    CONST robtarget p4016:= [[1554.6419767101188, 10.164661639834293, 993.500033578516], [0, 0, 1, 0], [0, 0, 0, 0], [9E9, 9E9, 9E9, 9E9, 9E9, 9E9]];
    CONST robtarget p4017:= [[1554.7008352009186, 9.837821442717242, 993.500033578516], [0, 0, 1, 0], [0, 0, 0, 0], [9E9, 9E9, 9E9, 9E9, 9E9, 9E9]];
    CONST robtarget p4018:= [[1554.7242404677872, 9.706052723327417, 993.500033578516], [0, 0, 1, 0], [0, 0, 0, 0], [9E9, 9E9, 9E9, 9E9, 9E9, 9E9]];
    CONST robtarget p4019:= [[1554.7649214276712, 9.482909780103284, 993.500033578516], [0, 0, 1, 0], [0, 0, 0, 0], [9E9, 9E9, 9E9, 9E9, 9E9, 9E9]];
    CONST robtarget p4020:= [[1554.8352270948067, 9.068291490106276, 993.500033578516], [0, 0, 1, 0], [0, 0, 0, 0], [9E9, 9E9, 9E9, 9E9, 9E9, 9E9]];
    CONST robtarget p4021:= [[1554.9212712484702, 8.59744226106804, 993.500033578516], [0, 0, 1, 0], [0, 0, 0, 0], [9E9, 9E9, 9E9, 9E9, 9E9, 9E9]];
    CONST robtarget p4022:= [[1555.0185066025715, 8.144599417769001, 993.500033578516], [0, 0, 1, 0], [0, 0, 0, 0], [9E9, 9E9, 9E9, 9E9, 9E9, 9E9]];
    CONST robtarget p4023:= [[1555.0385939462196, 7.9852680304157815, 993.500033578516], [0, 0, 1, 0], [0, 0, 0, 0], [9E9, 9E9, 9E9, 9E9, 9E9, 9E9]];
    CONST robtarget p4024:= [[1555.0668408502406, 7.720577334258238, 993.500033578516], [0, 0, 1, 0], [0, 0, 0, 0], [9E9, 9E9, 9E9, 9E9, 9E9, 9E9]];
    CONST robtarget p4025:= [[1555.1038402589074, 7.394988314848419, 993.500033578516], [0, 0, 1, 0], [0, 0, 0, 0], [9E9, 9E9, 9E9, 9E9, 9E9, 9E9]];
    CONST robtarget p4026:= [[1555.1141702872178, 7.2850707768797065, 993.500033578516], [0, 0, 1, 0], [0, 0, 0, 0], [9E9, 9E9, 9E9, 9E9, 9E9, 9E9]];
    CONST robtarget p4027:= [[1555.160055171739, 6.884447981356743, 993.500033578516], [0, 0, 1, 0], [0, 0, 0, 0], [9E9, 9E9, 9E9, 9E9, 9E9, 9E9]];
    CONST robtarget p4028:= [[1555.1886068304418, 6.5967447173674145, 993.500033578516], [0, 0, 1, 0], [0, 0, 0, 0], [9E9, 9E9, 9E9, 9E9, 9E9, 9E9]];
    CONST robtarget p4029:= [[1555.2302397704561, 6.209649884868298, 993.500033578516], [0, 0, 1, 0], [0, 0, 0, 0], [9E9, 9E9, 9E9, 9E9, 9E9, 9E9]];
    CONST robtarget p4030:= [[1555.3072534316846, 5.36442871184876, 993.500033578516], [0, 0, 1, 0], [0, 0, 0, 0], [9E9, 9E9, 9E9, 9E9, 9E9, 9E9]];
    CONST robtarget p4031:= [[1555.37826504701, 4.761405763737287, 993.500033578516], [0, 0, 1, 0], [0, 0, 0, 0], [9E9, 9E9, 9E9, 9E9, 9E9, 9E9]];
    CONST robtarget p4032:= [[1555.3863462726958, 4.670605801933405, 993.500033578516], [0, 0, 1, 0], [0, 0, 0, 0], [9E9, 9E9, 9E9, 9E9, 9E9, 9E9]];
    CONST robtarget p4033:= [[1555.4282420152724, 4.316200343407104, 993.500033578516], [0, 0, 1, 0], [0, 0, 0, 0], [9E9, 9E9, 9E9, 9E9, 9E9, 9E9]];
    CONST robtarget p4034:= [[1555.474795687078, 3.9231101854634716, 993.500033578516], [0, 0, 1, 0], [0, 0, 0, 0], [9E9, 9E9, 9E9, 9E9, 9E9, 9E9]];
    CONST robtarget p4035:= [[1555.4964332564984, 3.210495643507869, 993.500033578516], [0, 0, 1, 0], [0, 0, 0, 0], [9E9, 9E9, 9E9, 9E9, 9E9, 9E9]];
    CONST robtarget p4036:= [[1555.4992750024937, 3.001332927943622, 993.500033578516], [0, 0, 1, 0], [0, 0, 0, 0], [9E9, 9E9, 9E9, 9E9, 9E9, 9E9]];
    CONST robtarget p4037:= [[1555.5146870542724, 2.606860948282204, 993.500033578516], [0, 0, 1, 0], [0, 0, 0, 0], [9E9, 9E9, 9E9, 9E9, 9E9, 9E9]];
    CONST robtarget p4038:= [[1555.5401059955102, 2.158807079297702, 993.500033578516], [0, 0, 1, 0], [0, 0, 0, 0], [9E9, 9E9, 9E9, 9E9, 9E9, 9E9]];
    CONST robtarget p4039:= [[1555.5457042027897, 1.9240824141459996, 993.500033578516], [0, 0, 1, 0], [0, 0, 0, 0], [9E9, 9E9, 9E9, 9E9, 9E9, 9E9]];
    CONST robtarget p4040:= [[1555.5560129677121, 1.6442269998726573, 993.500033578516], [0, 0, 1, 0], [0, 0, 0, 0], [9E9, 9E9, 9E9, 9E9, 9E9, 9E9]];
    CONST robtarget p4041:= [[1555.5620302267785, 1.4813565941546756, 993.500033578516], [0, 0, 1, 0], [0, 0, 0, 0], [9E9, 9E9, 9E9, 9E9, 9E9, 9E9]];
    CONST robtarget p4042:= [[1555.569137398368, 1.3324889484946993, 993.500033578516], [0, 0, 1, 0], [0, 0, 0, 0], [9E9, 9E9, 9E9, 9E9, 9E9, 9E9]];
    CONST robtarget p4043:= [[1555.5836986010872, 0.9039823076832789, 993.500033578516], [0, 0, 1, 0], [0, 0, 0, 0], [9E9, 9E9, 9E9, 9E9, 9E9, 9E9]];
    CONST robtarget p4044:= [[1555.584302450153, 0.8259278887639994, 993.500033578516], [0, 0, 1, 0], [0, 0, 0, 0], [9E9, 9E9, 9E9, 9E9, 9E9, 9E9]];
    CONST robtarget p4045:= [[1555.5904849739145, 0.5579150837128566, 993.500033578516], [0, 0, 1, 0], [0, 0, 0, 0], [9E9, 9E9, 9E9, 9E9, 9E9, 9E9]];
    CONST robtarget p4046:= [[1555.6069058610203, 0.01192725742885159, 993.500033578516], [0, 0, 1, 0], [0, 0, 0, 0], [9E9, 9E9, 9E9, 9E9, 9E9, 9E9]];
    CONST robtarget p4047:= [[1555.6080018663752, -0.28272944407356704, 993.500033578516], [0, 0, 1, 0], [0, 0, 0, 0], [9E9, 9E9, 9E9, 9E9, 9E9, 9E9]];
    CONST robtarget p4048:= [[1555.5897069092575, -0.568370675110188, 993.500033578516], [0, 0, 1, 0], [0, 0, 0, 0], [9E9, 9E9, 9E9, 9E9, 9E9, 9E9]];
    CONST robtarget p4049:= [[1555.5753783303503, -1.0723405994250186, 993.500033578516], [0, 0, 1, 0], [0, 0, 0, 0], [9E9, 9E9, 9E9, 9E9, 9E9, 9E9]];
    CONST robtarget p4050:= [[1555.5457633836807, -1.5150721807046637, 993.500033578516], [0, 0, 1, 0], [0, 0, 0, 0], [9E9, 9E9, 9E9, 9E9, 9E9, 9E9]];
    CONST robtarget p4051:= [[1555.537896608749, -2.044805928378196, 993.500033578516], [0, 0, 1, 0], [0, 0, 0, 0], [9E9, 9E9, 9E9, 9E9, 9E9, 9E9]];
    CONST robtarget p4052:= [[1555.5215795409008, -2.3394641863057473, 993.500033578516], [0, 0, 1, 0], [0, 0, 0, 0], [9E9, 9E9, 9E9, 9E9, 9E9, 9E9]];
    CONST robtarget p4053:= [[1555.4995293223585, -2.83126276147442, 993.500033578516], [0, 0, 1, 0], [0, 0, 0, 0], [9E9, 9E9, 9E9, 9E9, 9E9, 9E9]];
    CONST robtarget p4054:= [[1555.500686212177, -3.2507572118477412, 993.500033578516], [0, 0, 1, 0], [0, 0, 0, 0], [9E9, 9E9, 9E9, 9E9, 9E9, 9E9]];
    CONST robtarget p4055:= [[1555.4801952520393, -3.540000238797006, 993.500033578516], [0, 0, 1, 0], [0, 0, 0, 0], [9E9, 9E9, 9E9, 9E9, 9E9, 9E9]];
    CONST robtarget p4056:= [[1555.475250706556, -3.909664977861297, 993.500033578516], [0, 0, 1, 0], [0, 0, 0, 0], [9E9, 9E9, 9E9, 9E9, 9E9, 9E9]];
    CONST robtarget p4057:= [[1555.4704758618002, -4.040117511451626, 993.500033578516], [0, 0, 1, 0], [0, 0, 0, 0], [9E9, 9E9, 9E9, 9E9, 9E9, 9E9]];
    CONST robtarget p4058:= [[1555.4548788143925, -4.184597877244968, 993.500033578516], [0, 0, 1, 0], [0, 0, 0, 0], [9E9, 9E9, 9E9, 9E9, 9E9, 9E9]];
    CONST robtarget p4059:= [[1555.3859897552957, -4.823125170682275, 993.500033578516], [0, 0, 1, 0], [0, 0, 0, 0], [9E9, 9E9, 9E9, 9E9, 9E9, 9E9]];
    CONST robtarget p4060:= [[1555.3511739675798, -5.082591974527546, 993.500033578516], [0, 0, 1, 0], [0, 0, 0, 0], [9E9, 9E9, 9E9, 9E9, 9E9, 9E9]];
    CONST robtarget p4061:= [[1555.3161022250322, -5.328723584463702, 993.500033578516], [0, 0, 1, 0], [0, 0, 0, 0], [9E9, 9E9, 9E9, 9E9, 9E9, 9E9]];
    CONST robtarget p4062:= [[1555.3021741428558, -5.461633220338783, 993.500033578516], [0, 0, 1, 0], [0, 0, 0, 0], [9E9, 9E9, 9E9, 9E9, 9E9, 9E9]];
    CONST robtarget p4063:= [[1555.2320437623023, -6.226398947024492, 993.500033578516], [0, 0, 1, 0], [0, 0, 0, 0], [9E9, 9E9, 9E9, 9E9, 9E9, 9E9]];
    CONST robtarget p4064:= [[1555.1608413042752, -6.821910992024904, 993.500033578516], [0, 0, 1, 0], [0, 0, 0, 0], [9E9, 9E9, 9E9, 9E9, 9E9, 9E9]];
    CONST robtarget p4065:= [[1555.1002904184656, -7.3310578421747365, 993.500033578516], [0, 0, 1, 0], [0, 0, 0, 0], [9E9, 9E9, 9E9, 9E9, 9E9, 9E9]];
    CONST robtarget p4066:= [[1555.075867870486, -7.565093083543573, 993.500033578516], [0, 0, 1, 0], [0, 0, 0, 0], [9E9, 9E9, 9E9, 9E9, 9E9, 9E9]];
    CONST robtarget p4067:= [[1555.0534446295678, -7.773617443065554, 993.500033578516], [0, 0, 1, 0], [0, 0, 0, 0], [9E9, 9E9, 9E9, 9E9, 9E9, 9E9]];
    CONST robtarget p4068:= [[1555.0292951011818, -8.048892820802436, 993.500033578516], [0, 0, 1, 0], [0, 0, 0, 0], [9E9, 9E9, 9E9, 9E9, 9E9, 9E9]];
    CONST robtarget p4069:= [[1555.000571435212, -8.20838796654671, 993.500033578516], [0, 0, 1, 0], [0, 0, 0, 0], [9E9, 9E9, 9E9, 9E9, 9E9, 9E9]];
    CONST robtarget p4070:= [[1554.9348620812655, -8.587526911211206, 993.500033578516], [0, 0, 1, 0], [0, 0, 0, 0], [9E9, 9E9, 9E9, 9E9, 9E9, 9E9]];
    CONST robtarget p4071:= [[1554.8414774526032, -9.07012225911049, 993.500033578516], [0, 0, 1, 0], [0, 0, 0, 0], [9E9, 9E9, 9E9, 9E9, 9E9, 9E9]];
    CONST robtarget p4072:= [[1554.7617777061982, -9.459953222433079, 993.500033578516], [0, 0, 1, 0], [0, 0, 0, 0], [9E9, 9E9, 9E9, 9E9, 9E9, 9E9]];
    CONST robtarget p4073:= [[1554.6532963114148, -9.950209852832828, 993.500033578516], [0, 0, 1, 0], [0, 0, 0, 0], [9E9, 9E9, 9E9, 9E9, 9E9, 9E9]];
    CONST robtarget p4074:= [[1554.5737452530968, -10.401613263807938, 993.500033578516], [0, 0, 1, 0], [0, 0, 0, 0], [9E9, 9E9, 9E9, 9E9, 9E9, 9E9]];
    CONST robtarget p4075:= [[1554.5310032922928, -10.744261336840545, 993.500033578516], [0, 0, 1, 0], [0, 0, 0, 0], [9E9, 9E9, 9E9, 9E9, 9E9, 9E9]];
    CONST robtarget p4076:= [[1554.4848696641359, -10.996810355268067, 993.500033578516], [0, 0, 1, 0], [0, 0, 0, 0], [9E9, 9E9, 9E9, 9E9, 9E9, 9E9]];
    CONST robtarget p4077:= [[1554.429524387338, -11.293607711081144, 993.500033578516], [0, 0, 1, 0], [0, 0, 0, 0], [9E9, 9E9, 9E9, 9E9, 9E9, 9E9]];
    CONST robtarget p4078:= [[1554.365244509884, -11.681877794735506, 993.500033578516], [0, 0, 1, 0], [0, 0, 0, 0], [9E9, 9E9, 9E9, 9E9, 9E9, 9E9]];
    CONST robtarget p4079:= [[1554.260654796157, -12.196206477131277, 993.500033578516], [0, 0, 1, 0], [0, 0, 0, 0], [9E9, 9E9, 9E9, 9E9, 9E9, 9E9]];
    CONST robtarget p4080:= [[1554.0305975482188, -13.054502339188467, 993.500033578516], [0, 0, 1, 0], [0, 0, 0, 0], [9E9, 9E9, 9E9, 9E9, 9E9, 9E9]];
    CONST robtarget p4081:= [[1553.977430038342, -13.263407594856204, 993.500033578516], [0, 0, 1, 0], [0, 0, 0, 0], [9E9, 9E9, 9E9, 9E9, 9E9, 9E9]];
    CONST robtarget p4082:= [[1553.85597144588, -13.716347986773343, 993.500033578516], [0, 0, 1, 0], [0, 0, 0, 0], [9E9, 9E9, 9E9, 9E9, 9E9, 9E9]];
    CONST robtarget p4083:= [[1553.735275178501, -14.166553581183678, 993.500033578516], [0, 0, 1, 0], [0, 0, 0, 0], [9E9, 9E9, 9E9, 9E9, 9E9, 9E9]];
    CONST robtarget p4084:= [[1553.7003844703927, -14.311016881022638, 993.500033578516], [0, 0, 1, 0], [0, 0, 0, 0], [9E9, 9E9, 9E9, 9E9, 9E9, 9E9]];
    CONST robtarget p4085:= [[1553.645211788333, -14.53618350036087, 993.500033578516], [0, 0, 1, 0], [0, 0, 0, 0], [9E9, 9E9, 9E9, 9E9, 9E9, 9E9]];
    CONST robtarget p4086:= [[1553.6005708615592, -14.710812405265642, 993.500033578516], [0, 0, 1, 0], [0, 0, 0, 0], [9E9, 9E9, 9E9, 9E9, 9E9, 9E9]];
    CONST robtarget p4087:= [[1553.4680572597388, -15.164164355499594, 993.500033578516], [0, 0, 1, 0], [0, 0, 0, 0], [9E9, 9E9, 9E9, 9E9, 9E9, 9E9]];
    CONST robtarget p4088:= [[1553.3773848306819, -15.536258371461692, 993.500033578516], [0, 0, 1, 0], [0, 0, 0, 0], [9E9, 9E9, 9E9, 9E9, 9E9, 9E9]];
    CONST robtarget p4089:= [[1553.2735747687145, -15.922966612214687, 993.500033578516], [0, 0, 1, 0], [0, 0, 0, 0], [9E9, 9E9, 9E9, 9E9, 9E9, 9E9]];
    CONST robtarget p4090:= [[1553.1492330594576, -16.30415940387421, 993.500033578516], [0, 0, 1, 0], [0, 0, 0, 0], [9E9, 9E9, 9E9, 9E9, 9E9, 9E9]];
    CONST robtarget p4091:= [[1553.1068559586142, -16.437841935749276, 993.500033578516], [0, 0, 1, 0], [0, 0, 0, 0], [9E9, 9E9, 9E9, 9E9, 9E9, 9E9]];
    CONST robtarget p4092:= [[1552.9948033201092, -16.80437930612829, 993.500033578516], [0, 0, 1, 0], [0, 0, 0, 0], [9E9, 9E9, 9E9, 9E9, 9E9, 9E9]];
    CONST robtarget p4093:= [[1552.824638434181, -17.29095365638217, 993.500033578516], [0, 0, 1, 0], [0, 0, 0, 0], [9E9, 9E9, 9E9, 9E9, 9E9, 9E9]];
    CONST robtarget p4094:= [[1552.6743421326719, -17.695280477599724, 993.500033578516], [0, 0, 1, 0], [0, 0, 0, 0], [9E9, 9E9, 9E9, 9E9, 9E9, 9E9]];
    CONST robtarget p4095:= [[1552.5185312246495, -18.18205253138484, 993.500033578516], [0, 0, 1, 0], [0, 0, 0, 0], [9E9, 9E9, 9E9, 9E9, 9E9, 9E9]];
    CONST robtarget p4096:= [[1552.430217919832, -18.42750320420714, 993.500033578516], [0, 0, 1, 0], [0, 0, 0, 0], [9E9, 9E9, 9E9, 9E9, 9E9, 9E9]];
    CONST robtarget p4097:= [[1552.1579420833923, -19.24711499655084, 993.500033578516], [0, 0, 1, 0], [0, 0, 0, 0], [9E9, 9E9, 9E9, 9E9, 9E9, 9E9]];
    CONST robtarget p4098:= [[1551.9948060843485, -19.723002973923855, 993.500033578516], [0, 0, 1, 0], [0, 0, 0, 0], [9E9, 9E9, 9E9, 9E9, 9E9, 9E9]];
    CONST robtarget p4099:= [[1551.9764390452037, -19.78836428857487, 993.500033578516], [0, 0, 1, 0], [0, 0, 0, 0], [9E9, 9E9, 9E9, 9E9, 9E9, 9E9]];
    CONST robtarget p4100:= [[1551.77860658663, -20.25262789073657, 993.500033578516], [0, 0, 1, 0], [0, 0, 0, 0], [9E9, 9E9, 9E9, 9E9, 9E9, 9E9]];
    CONST robtarget p4101:= [[1551.732954511871, -20.36336320736133, 993.500033578516], [0, 0, 1, 0], [0, 0, 0, 0], [9E9, 9E9, 9E9, 9E9, 9E9, 9E9]];
    CONST robtarget p4102:= [[1551.4159413272039, -21.11609605269785, 993.500033578516], [0, 0, 1, 0], [0, 0, 0, 0], [9E9, 9E9, 9E9, 9E9, 9E9, 9E9]];
    CONST robtarget p4103:= [[1551.3366522843414, -21.304909789410537, 993.500033578516], [0, 0, 1, 0], [0, 0, 0, 0], [9E9, 9E9, 9E9, 9E9, 9E9, 9E9]];
    CONST robtarget p4104:= [[1551.1988748219385, -21.630752784024033, 993.500033578516], [0, 0, 1, 0], [0, 0, 0, 0], [9E9, 9E9, 9E9, 9E9, 9E9, 9E9]];
    CONST robtarget p4105:= [[1551.115064733889, -21.821661267412765, 993.500033578516], [0, 0, 1, 0], [0, 0, 0, 0], [9E9, 9E9, 9E9, 9E9, 9E9, 9E9]];
    CONST robtarget p4106:= [[1551.0637969386862, -21.926989670457786, 993.500033578516], [0, 0, 1, 0], [0, 0, 0, 0], [9E9, 9E9, 9E9, 9E9, 9E9, 9E9]];
    CONST robtarget p4107:= [[1550.8234789540143, -22.48761161410414, 993.500033578516], [0, 0, 1, 0], [0, 0, 0, 0], [9E9, 9E9, 9E9, 9E9, 9E9, 9E9]];
    CONST robtarget p4108:= [[1550.7416655792576, -22.70735182238834, 993.500033578516], [0, 0, 1, 0], [0, 0, 0, 0], [9E9, 9E9, 9E9, 9E9, 9E9, 9E9]];
    CONST robtarget p4109:= [[1550.5373248839085, -23.179126462561022, 993.500033578516], [0, 0, 1, 0], [0, 0, 0, 0], [9E9, 9E9, 9E9, 9E9, 9E9, 9E9]];
    CONST robtarget p4110:= [[1550.3466691258116, -23.632344017919024, 993.500033578516], [0, 0, 1, 0], [0, 0, 0, 0], [9E9, 9E9, 9E9, 9E9, 9E9, 9E9]];
    CONST robtarget p4111:= [[1550.3255378976685, -23.675425425283905, 993.500033578516], [0, 0, 1, 0], [0, 0, 0, 0], [9E9, 9E9, 9E9, 9E9, 9E9, 9E9]];
    CONST robtarget p4112:= [[1550.181348683183, -23.946530709164044, 993.500033578516], [0, 0, 1, 0], [0, 0, 0, 0], [9E9, 9E9, 9E9, 9E9, 9E9, 9E9]];
    CONST robtarget p4113:= [[1550.044079598348, -24.21167120523466, 993.500033578516], [0, 0, 1, 0], [0, 0, 0, 0], [9E9, 9E9, 9E9, 9E9, 9E9, 9E9]];
    CONST robtarget p4114:= [[1549.8514748131022, -24.548156501795795, 993.500033578516], [0, 0, 1, 0], [0, 0, 0, 0], [9E9, 9E9, 9E9, 9E9, 9E9, 9E9]];
    CONST robtarget p4115:= [[1549.5804014377222, -25.124889272529053, 993.500033578516], [0, 0, 1, 0], [0, 0, 0, 0], [9E9, 9E9, 9E9, 9E9, 9E9, 9E9]];
    CONST robtarget p4116:= [[1549.5405593055677, -25.20439410297127, 993.500033578516], [0, 0, 1, 0], [0, 0, 0, 0], [9E9, 9E9, 9E9, 9E9, 9E9, 9E9]];
    CONST robtarget p4117:= [[1549.3456798913373, -25.577151773368456, 993.500033578516], [0, 0, 1, 0], [0, 0, 0, 0], [9E9, 9E9, 9E9, 9E9, 9E9, 9E9]];
    CONST robtarget p4118:= [[1549.0329507630183, -26.171345531936993, 993.500033578516], [0, 0, 1, 0], [0, 0, 0, 0], [9E9, 9E9, 9E9, 9E9, 9E9, 9E9]];
    CONST robtarget p4119:= [[1548.9223972633604, -26.36387979337215, 993.500033578516], [0, 0, 1, 0], [0, 0, 0, 0], [9E9, 9E9, 9E9, 9E9, 9E9, 9E9]];
    CONST robtarget p4120:= [[1548.730649815, -26.733301295106727, 993.500033578516], [0, 0, 1, 0], [0, 0, 0, 0], [9E9, 9E9, 9E9, 9E9, 9E9, 9E9]];
    CONST robtarget p4121:= [[1548.5590267187338, -27.109148307826146, 993.500033578516], [0, 0, 1, 0], [0, 0, 0, 0], [9E9, 9E9, 9E9, 9E9, 9E9, 9E9]];
    CONST robtarget p4122:= [[1548.3443713859592, -27.4625186247931, 993.500033578516], [0, 0, 1, 0], [0, 0, 0, 0], [9E9, 9E9, 9E9, 9E9, 9E9, 9E9]];
    CONST robtarget p4123:= [[1548.0588032035475, -27.95023195473138, 993.500033578516], [0, 0, 1, 0], [0, 0, 0, 0], [9E9, 9E9, 9E9, 9E9, 9E9, 9E9]];
    CONST robtarget p4124:= [[1547.9119052588649, -28.178025883520945, 993.500033578516], [0, 0, 1, 0], [0, 0, 0, 0], [9E9, 9E9, 9E9, 9E9, 9E9, 9E9]];
    CONST robtarget p4125:= [[1547.7246936658817, -28.471151096174346, 993.500033578516], [0, 0, 1, 0], [0, 0, 0, 0], [9E9, 9E9, 9E9, 9E9, 9E9, 9E9]];
    CONST robtarget p4126:= [[1547.4806495127852, -28.888958116495914, 993.500033578516], [0, 0, 1, 0], [0, 0, 0, 0], [9E9, 9E9, 9E9, 9E9, 9E9, 9E9]];
    CONST robtarget p4127:= [[1547.1593093200343, -29.39622454088626, 993.500033578516], [0, 0, 1, 0], [0, 0, 0, 0], [9E9, 9E9, 9E9, 9E9, 9E9, 9E9]];
    CONST robtarget p4128:= [[1547.0482572291721, -29.602114632359836, 993.500033578516], [0, 0, 1, 0], [0, 0, 0, 0], [9E9, 9E9, 9E9, 9E9, 9E9, 9E9]];
    CONST robtarget p4129:= [[1546.6316299331197, -30.277961389395664, 993.500033578516], [0, 0, 1, 0], [0, 0, 0, 0], [9E9, 9E9, 9E9, 9E9, 9E9, 9E9]];
    CONST robtarget p4130:= [[1546.5916573944664, -30.348003455662123, 993.500033578516], [0, 0, 1, 0], [0, 0, 0, 0], [9E9, 9E9, 9E9, 9E9, 9E9, 9E9]];
    CONST robtarget p4131:= [[1546.5392322795406, -30.429748980631025, 993.500033578516], [0, 0, 1, 0], [0, 0, 0, 0], [9E9, 9E9, 9E9, 9E9, 9E9, 9E9]];
    CONST robtarget p4132:= [[1546.3678912033913, -30.682996185938215, 993.500033578516], [0, 0, 1, 0], [0, 0, 0, 0], [9E9, 9E9, 9E9, 9E9, 9E9, 9E9]];
    CONST robtarget p4133:= [[1546.3215018780127, -30.753596904321526, 993.500033578516], [0, 0, 1, 0], [0, 0, 0, 0], [9E9, 9E9, 9E9, 9E9, 9E9, 9E9]];
    CONST robtarget p4134:= [[1546.1580669226219, -30.9898374185305, 993.500033578516], [0, 0, 1, 0], [0, 0, 0, 0], [9E9, 9E9, 9E9, 9E9, 9E9, 9E9]];
    CONST robtarget p4135:= [[1546.126538337522, -31.034846710935234, 993.500033578516], [0, 0, 1, 0], [0, 0, 0, 0], [9E9, 9E9, 9E9, 9E9, 9E9, 9E9]];
    CONST robtarget p4136:= [[1545.9442168653484, -31.30068098401418, 993.500033578516], [0, 0, 1, 0], [0, 0, 0, 0], [9E9, 9E9, 9E9, 9E9, 9E9, 9E9]];
    CONST robtarget p4137:= [[1545.916904883265, -31.33684404044449, 993.500033578516], [0, 0, 1, 0], [0, 0, 0, 0], [9E9, 9E9, 9E9, 9E9, 9E9, 9E9]];
    CONST robtarget p4138:= [[1545.7163208127422, -31.621902815478954, 993.500033578516], [0, 0, 1, 0], [0, 0, 0, 0], [9E9, 9E9, 9E9, 9E9, 9E9, 9E9]];
    CONST robtarget p4139:= [[1545.3617400820876, -32.081262731677334, 993.500033578516], [0, 0, 1, 0], [0, 0, 0, 0], [9E9, 9E9, 9E9, 9E9, 9E9, 9E9]];
    CONST robtarget p4140:= [[1545.2095973541207, -32.316530430876554, 993.500033578516], [0, 0, 1, 0], [0, 0, 0, 0], [9E9, 9E9, 9E9, 9E9, 9E9, 9E9]];
    CONST robtarget p4141:= [[1545.1416000154663, -32.42271351780253, 993.500033578516], [0, 0, 1, 0], [0, 0, 0, 0], [9E9, 9E9, 9E9, 9E9, 9E9, 9E9]];
    CONST robtarget p4142:= [[1545.007174085452, -32.61646527440308, 993.500033578516], [0, 0, 1, 0], [0, 0, 0, 0], [9E9, 9E9, 9E9, 9E9, 9E9, 9E9]];
    CONST robtarget p4143:= [[1544.6852272392653, -33.04443502943098, 993.500033578516], [0, 0, 1, 0], [0, 0, 0, 0], [9E9, 9E9, 9E9, 9E9, 9E9, 9E9]];
    CONST robtarget p4144:= [[1544.3078520840118, -33.57971848815495, 993.500033578516], [0, 0, 1, 0], [0, 0, 0, 0], [9E9, 9E9, 9E9, 9E9, 9E9, 9E9]];
    CONST robtarget p4145:= [[1544.2293677667458, -33.69470874185417, 993.500033578516], [0, 0, 1, 0], [0, 0, 0, 0], [9E9, 9E9, 9E9, 9E9, 9E9, 9E9]];
    CONST robtarget p4146:= [[1544.061613706892, -33.938863462766435, 993.500033578516], [0, 0, 1, 0], [0, 0, 0, 0], [9E9, 9E9, 9E9, 9E9, 9E9, 9E9]];
    CONST robtarget p4147:= [[1544.0063296445308, -34.015018154159776, 993.500033578516], [0, 0, 1, 0], [0, 0, 0, 0], [9E9, 9E9, 9E9, 9E9, 9E9, 9E9]];
    CONST robtarget p4148:= [[1543.4194648245095, -34.72085352168525, 993.500033578516], [0, 0, 1, 0], [0, 0, 0, 0], [9E9, 9E9, 9E9, 9E9, 9E9, 9E9]];
    CONST robtarget p4149:= [[1543.1490701329767, -35.04086372199627, 993.500033578516], [0, 0, 1, 0], [0, 0, 0, 0], [9E9, 9E9, 9E9, 9E9, 9E9, 9E9]];
    CONST robtarget p4150:= [[1542.9764648879466, -35.24299878117947, 993.500033578516], [0, 0, 1, 0], [0, 0, 0, 0], [9E9, 9E9, 9E9, 9E9, 9E9, 9E9]];
    CONST robtarget p4151:= [[1542.8976099171116, -35.335683321207526, 993.500033578516], [0, 0, 1, 0], [0, 0, 0, 0], [9E9, 9E9, 9E9, 9E9, 9E9, 9E9]];
    CONST robtarget p4152:= [[1542.686811608819, -35.593294239601285, 993.500033578516], [0, 0, 1, 0], [0, 0, 0, 0], [9E9, 9E9, 9E9, 9E9, 9E9, 9E9]];
    CONST robtarget p4153:= [[1542.533440167045, -35.762068528757226, 993.500033578516], [0, 0, 1, 0], [0, 0, 0, 0], [9E9, 9E9, 9E9, 9E9, 9E9, 9E9]];
    CONST robtarget p4154:= [[1542.2771647721138, -36.06563167221814, 993.500033578516], [0, 0, 1, 0], [0, 0, 0, 0], [9E9, 9E9, 9E9, 9E9, 9E9, 9E9]];
    CONST robtarget p4155:= [[1542.0642130642232, -36.3374435672405, 993.500033578516], [0, 0, 1, 0], [0, 0, 0, 0], [9E9, 9E9, 9E9, 9E9, 9E9, 9E9]];
    CONST robtarget p4156:= [[1541.7474803894224, -36.724880336206766, 993.500033578516], [0, 0, 1, 0], [0, 0, 0, 0], [9E9, 9E9, 9E9, 9E9, 9E9, 9E9]];
    CONST robtarget p4157:= [[1541.626708731916, -36.87241836739917, 993.500033578516], [0, 0, 1, 0], [0, 0, 0, 0], [9E9, 9E9, 9E9, 9E9, 9E9, 9E9]];
    CONST robtarget p4158:= [[1541.4723368843722, -37.0518217399505, 993.500033578516], [0, 0, 1, 0], [0, 0, 0, 0], [9E9, 9E9, 9E9, 9E9, 9E9, 9E9]];
    CONST robtarget p4159:= [[1541.2637566089825, -37.27995852886669, 993.500033578516], [0, 0, 1, 0], [0, 0, 0, 0], [9E9, 9E9, 9E9, 9E9, 9E9, 9E9]];
    CONST robtarget p4160:= [[1541.1343961680013, -37.41609395445425, 993.500033578516], [0, 0, 1, 0], [0, 0, 0, 0], [9E9, 9E9, 9E9, 9E9, 9E9, 9E9]];
    CONST robtarget p4161:= [[1540.9620780620705, -37.58167845975497, 993.500033578516], [0, 0, 1, 0], [0, 0, 0, 0], [9E9, 9E9, 9E9, 9E9, 9E9, 9E9]];
    CONST robtarget p4162:= [[1540.737647725568, -37.81054650436012, 993.500033578516], [0, 0, 1, 0], [0, 0, 0, 0], [9E9, 9E9, 9E9, 9E9, 9E9, 9E9]];
    CONST robtarget p4163:= [[1540.4518972325213, -38.10761777096063, 993.500033578516], [0, 0, 1, 0], [0, 0, 0, 0], [9E9, 9E9, 9E9, 9E9, 9E9, 9E9]];
    CONST robtarget p4164:= [[1540.3258726021872, -38.25138599808624, 993.500033578516], [0, 0, 1, 0], [0, 0, 0, 0], [9E9, 9E9, 9E9, 9E9, 9E9, 9E9]];
    CONST robtarget p4165:= [[1540.221959710798, -38.364241979095375, 993.500033578516], [0, 0, 1, 0], [0, 0, 0, 0], [9E9, 9E9, 9E9, 9E9, 9E9, 9E9]];
    CONST robtarget p4166:= [[1540.0310396601287, -38.56067181755926, 993.500033578516], [0, 0, 1, 0], [0, 0, 0, 0], [9E9, 9E9, 9E9, 9E9, 9E9, 9E9]];
    CONST robtarget p4167:= [[1539.5383119060127, -39.07227979513109, 993.500033578516], [0, 0, 1, 0], [0, 0, 0, 0], [9E9, 9E9, 9E9, 9E9, 9E9, 9E9]];
    CONST robtarget p4168:= [[1539.3609513649412, -39.25314710575125, 993.500033578516], [0, 0, 1, 0], [0, 0, 0, 0], [9E9, 9E9, 9E9, 9E9, 9E9, 9E9]];
    CONST robtarget p4169:= [[1538.9526282731272, -39.66410900769987, 993.500033578516], [0, 0, 1, 0], [0, 0, 0, 0], [9E9, 9E9, 9E9, 9E9, 9E9, 9E9]];
    CONST robtarget p4170:= [[1538.7310081810106, -39.89796970277656, 993.500033578516], [0, 0, 1, 0], [0, 0, 0, 0], [9E9, 9E9, 9E9, 9E9, 9E9, 9E9]];
    CONST robtarget p4171:= [[1538.6823680020225, -39.94219119540354, 993.500033578516], [0, 0, 1, 0], [0, 0, 0, 0], [9E9, 9E9, 9E9, 9E9, 9E9, 9E9]];
    CONST robtarget p4172:= [[1538.1671502889121, -40.39412755043739, 993.500033578516], [0, 0, 1, 0], [0, 0, 0, 0], [9E9, 9E9, 9E9, 9E9, 9E9, 9E9]];
    CONST robtarget p4173:= [[1537.7426660821727, -40.806788619232634, 993.500033578516], [0, 0, 1, 0], [0, 0, 0, 0], [9E9, 9E9, 9E9, 9E9, 9E9, 9E9]];
    CONST robtarget p4174:= [[1537.6928287305013, -40.85672083744086, 993.500033578516], [0, 0, 1, 0], [0, 0, 0, 0], [9E9, 9E9, 9E9, 9E9, 9E9, 9E9]];
    CONST robtarget p4175:= [[1537.3793899639877, -41.12348194719298, 993.500033578516], [0, 0, 1, 0], [0, 0, 0, 0], [9E9, 9E9, 9E9, 9E9, 9E9, 9E9]];
    CONST robtarget p4176:= [[1537.12938588905, -41.343663537613374, 993.500033578516], [0, 0, 1, 0], [0, 0, 0, 0], [9E9, 9E9, 9E9, 9E9, 9E9, 9E9]];
    CONST robtarget p4177:= [[1536.902774382986, -41.55007312660826, 993.500033578516], [0, 0, 1, 0], [0, 0, 0, 0], [9E9, 9E9, 9E9, 9E9, 9E9, 9E9]];
    CONST robtarget p4178:= [[1536.7167131016504, -41.731288804072726, 993.500033578516], [0, 0, 1, 0], [0, 0, 0, 0], [9E9, 9E9, 9E9, 9E9, 9E9, 9E9]];
    CONST robtarget p4179:= [[1536.532935866802, -41.8901835897854, 993.500033578516], [0, 0, 1, 0], [0, 0, 0, 0], [9E9, 9E9, 9E9, 9E9, 9E9, 9E9]];
    CONST robtarget p4180:= [[1536.1608934437356, -42.21572078222415, 993.500033578516], [0, 0, 1, 0], [0, 0, 0, 0], [9E9, 9E9, 9E9, 9E9, 9E9, 9E9]];
    CONST robtarget p4181:= [[1536.1233677565858, -42.24708255215591, 993.500033578516], [0, 0, 1, 0], [0, 0, 0, 0], [9E9, 9E9, 9E9, 9E9, 9E9, 9E9]];
    CONST robtarget p4182:= [[1535.730685183453, -42.58714623648291, 993.500033578516], [0, 0, 1, 0], [0, 0, 0, 0], [9E9, 9E9, 9E9, 9E9, 9E9, 9E9]];
    CONST robtarget p4183:= [[1535.6604397826175, -42.65149110961505, 993.500033578516], [0, 0, 1, 0], [0, 0, 0, 0], [9E9, 9E9, 9E9, 9E9, 9E9, 9E9]];
    CONST robtarget p4184:= [[1535.2893823465506, -42.95375005674663, 993.500033578516], [0, 0, 1, 0], [0, 0, 0, 0], [9E9, 9E9, 9E9, 9E9, 9E9, 9E9]];
    CONST robtarget p4185:= [[1535.190048337098, -43.03657610010355, 993.500033578516], [0, 0, 1, 0], [0, 0, 0, 0], [9E9, 9E9, 9E9, 9E9, 9E9, 9E9]];
    CONST robtarget p4186:= [[1534.9087409060442, -43.26802889781054, 993.500033578516], [0, 0, 1, 0], [0, 0, 0, 0], [9E9, 9E9, 9E9, 9E9, 9E9, 9E9]];
    CONST robtarget p4187:= [[1534.6227849700576, -43.489716754368956, 993.500033578516], [0, 0, 1, 0], [0, 0, 0, 0], [9E9, 9E9, 9E9, 9E9, 9E9, 9E9]];
    CONST robtarget p4188:= [[1534.2772620596647, -43.75409785421051, 993.500033578516], [0, 0, 1, 0], [0, 0, 0, 0], [9E9, 9E9, 9E9, 9E9, 9E9, 9E9]];
    CONST robtarget p4189:= [[1533.731225645397, -44.17898602822898, 993.500033578516], [0, 0, 1, 0], [0, 0, 0, 0], [9E9, 9E9, 9E9, 9E9, 9E9, 9E9]];
    CONST robtarget p4190:= [[1533.3486991712523, -44.47333364915849, 993.500033578516], [0, 0, 1, 0], [0, 0, 0, 0], [9E9, 9E9, 9E9, 9E9, 9E9, 9E9]];
    CONST robtarget p4191:= [[1533.1698965289236, -44.611141714070854, 993.500033578516], [0, 0, 1, 0], [0, 0, 0, 0], [9E9, 9E9, 9E9, 9E9, 9E9, 9E9]];
    CONST robtarget p4192:= [[1532.5699672005803, -45.04577386468151, 993.500033578516], [0, 0, 1, 0], [0, 0, 0, 0], [9E9, 9E9, 9E9, 9E9, 9E9, 9E9]];
    CONST robtarget p4193:= [[1532.3285414352222, -45.24262827224148, 993.500033578516], [0, 0, 1, 0], [0, 0, 0, 0], [9E9, 9E9, 9E9, 9E9, 9E9, 9E9]];
    CONST robtarget p4194:= [[1532.1711269768564, -45.350240987288196, 993.500033578516], [0, 0, 1, 0], [0, 0, 0, 0], [9E9, 9E9, 9E9, 9E9, 9E9, 9E9]];
    CONST robtarget p4195:= [[1531.8011306779201, -45.600780745273966, 993.500033578516], [0, 0, 1, 0], [0, 0, 0, 0], [9E9, 9E9, 9E9, 9E9, 9E9, 9E9]];
    CONST robtarget p4196:= [[1531.3696493100233, -45.89533481680043, 993.500033578516], [0, 0, 1, 0], [0, 0, 0, 0], [9E9, 9E9, 9E9, 9E9, 9E9, 9E9]];
    CONST robtarget p4197:= [[1530.8718958306054, -46.2235979997289, 993.500033578516], [0, 0, 1, 0], [0, 0, 0, 0], [9E9, 9E9, 9E9, 9E9, 9E9, 9E9]];
    CONST robtarget p4198:= [[1530.4171827602966, -46.519819219502665, 993.500033578516], [0, 0, 1, 0], [0, 0, 0, 0], [9E9, 9E9, 9E9, 9E9, 9E9, 9E9]];
    CONST robtarget p4199:= [[1530.217263460704, -46.65507793694422, 993.500033578516], [0, 0, 1, 0], [0, 0, 0, 0], [9E9, 9E9, 9E9, 9E9, 9E9, 9E9]];
    CONST robtarget p4200:= [[1530.056746301974, -46.763916023469164, 993.500033578516], [0, 0, 1, 0], [0, 0, 0, 0], [9E9, 9E9, 9E9, 9E9, 9E9, 9E9]];
    CONST robtarget p4201:= [[1529.843456974275, -46.89478531411835, 993.500033578516], [0, 0, 1, 0], [0, 0, 0, 0], [9E9, 9E9, 9E9, 9E9, 9E9, 9E9]];
    CONST robtarget p4202:= [[1529.5449194374721, -47.08894844573004, 993.500033578516], [0, 0, 1, 0], [0, 0, 0, 0], [9E9, 9E9, 9E9, 9E9, 9E9, 9E9]];
    CONST robtarget p4203:= [[1529.342945411055, -47.21777771435845, 993.500033578516], [0, 0, 1, 0], [0, 0, 0, 0], [9E9, 9E9, 9E9, 9E9, 9E9, 9E9]];
    CONST robtarget p4204:= [[1529.2642628061528, -47.26845116210754, 993.500033578516], [0, 0, 1, 0], [0, 0, 0, 0], [9E9, 9E9, 9E9, 9E9, 9E9, 9E9]];
    CONST robtarget p4205:= [[1528.9606171375442, -47.46000468829058, 993.500033578516], [0, 0, 1, 0], [0, 0, 0, 0], [9E9, 9E9, 9E9, 9E9, 9E9, 9E9]];
    CONST robtarget p4206:= [[1528.854017059838, -47.53240555719428, 993.500033578516], [0, 0, 1, 0], [0, 0, 0, 0], [9E9, 9E9, 9E9, 9E9, 9E9, 9E9]];
    CONST robtarget p4207:= [[1528.7572243049733, -47.60115890079086, 993.500033578516], [0, 0, 1, 0], [0, 0, 0, 0], [9E9, 9E9, 9E9, 9E9, 9E9, 9E9]];
    CONST robtarget p4208:= [[1528.2472190530716, -47.87224657471093, 993.500033578516], [0, 0, 1, 0], [0, 0, 0, 0], [9E9, 9E9, 9E9, 9E9, 9E9, 9E9]];
    CONST robtarget p4209:= [[1528.089723356518, -47.96046687107399, 993.500033578516], [0, 0, 1, 0], [0, 0, 0, 0], [9E9, 9E9, 9E9, 9E9, 9E9, 9E9]];
    CONST robtarget p4210:= [[1527.7613737518932, -48.16042821606706, 993.500033578516], [0, 0, 1, 0], [0, 0, 0, 0], [9E9, 9E9, 9E9, 9E9, 9E9, 9E9]];
    CONST robtarget p4211:= [[1527.4223317010822, -48.336459807540216, 993.500033578516], [0, 0, 1, 0], [0, 0, 0, 0], [9E9, 9E9, 9E9, 9E9, 9E9, 9E9]];
    CONST robtarget p4212:= [[1527.1537893921482, -48.49569041285845, 993.500033578516], [0, 0, 1, 0], [0, 0, 0, 0], [9E9, 9E9, 9E9, 9E9, 9E9, 9E9]];
    CONST robtarget p4213:= [[1526.6622117105692, -48.766884964356855, 993.500033578516], [0, 0, 1, 0], [0, 0, 0, 0], [9E9, 9E9, 9E9, 9E9, 9E9, 9E9]];
    CONST robtarget p4214:= [[1526.0238858030477, -49.12127030415674, 993.500033578516], [0, 0, 1, 0], [0, 0, 0, 0], [9E9, 9E9, 9E9, 9E9, 9E9, 9E9]];
    CONST robtarget p4215:= [[1525.7574801177627, -49.2773840187095, 993.500033578516], [0, 0, 1, 0], [0, 0, 0, 0], [9E9, 9E9, 9E9, 9E9, 9E9, 9E9]];
    CONST robtarget p4216:= [[1525.577882863274, -49.37973856644577, 993.500033578516], [0, 0, 1, 0], [0, 0, 0, 0], [9E9, 9E9, 9E9, 9E9, 9E9, 9E9]];
    CONST robtarget p4217:= [[1525.2237205693089, -49.561652839755894, 993.500033578516], [0, 0, 1, 0], [0, 0, 0, 0], [9E9, 9E9, 9E9, 9E9, 9E9, 9E9]];
    CONST robtarget p4218:= [[1524.926271596964, -49.69541940584739, 993.500033578516], [0, 0, 1, 0], [0, 0, 0, 0], [9E9, 9E9, 9E9, 9E9, 9E9, 9E9]];
    CONST robtarget p4219:= [[1524.7015967810225, -49.78951989434897, 993.500033578516], [0, 0, 1, 0], [0, 0, 0, 0], [9E9, 9E9, 9E9, 9E9, 9E9, 9E9]];
    CONST robtarget p4220:= [[1524.1525739605709, -50.044907571137315, 993.500033578516], [0, 0, 1, 0], [0, 0, 0, 0], [9E9, 9E9, 9E9, 9E9, 9E9, 9E9]];
    CONST robtarget p4221:= [[1523.8837359155798, -50.19095617833235, 993.500033578516], [0, 0, 1, 0], [0, 0, 0, 0], [9E9, 9E9, 9E9, 9E9, 9E9, 9E9]];
    CONST robtarget p4222:= [[1523.4553888288974, -50.383361753387604, 993.500033578516], [0, 0, 1, 0], [0, 0, 0, 0], [9E9, 9E9, 9E9, 9E9, 9E9, 9E9]];
    CONST robtarget p4223:= [[1523.3143739031275, -50.455270994846735, 993.500033578516], [0, 0, 1, 0], [0, 0, 0, 0], [9E9, 9E9, 9E9, 9E9, 9E9, 9E9]];
    CONST robtarget p4224:= [[1522.9391457413753, -50.62815142759504, 993.500033578516], [0, 0, 1, 0], [0, 0, 0, 0], [9E9, 9E9, 9E9, 9E9, 9E9, 9E9]];
    CONST robtarget p4225:= [[1522.9203013809442, -50.635442420488644, 993.500033578516], [0, 0, 1, 0], [0, 0, 0, 0], [9E9, 9E9, 9E9, 9E9, 9E9, 9E9]];
    CONST robtarget p4226:= [[1522.3452019789422, -50.89091936188008, 993.500033578516], [0, 0, 1, 0], [0, 0, 0, 0], [9E9, 9E9, 9E9, 9E9, 9E9, 9E9]];
    CONST robtarget p4227:= [[1522.036836918105, -51.054106002755084, 993.500033578516], [0, 0, 1, 0], [0, 0, 0, 0], [9E9, 9E9, 9E9, 9E9, 9E9, 9E9]];
    CONST robtarget p4228:= [[1521.5777112698881, -51.2571224485676, 993.500033578516], [0, 0, 1, 0], [0, 0, 0, 0], [9E9, 9E9, 9E9, 9E9, 9E9, 9E9]];
    CONST robtarget p4229:= [[1521.3787500024446, -51.330769902801805, 993.500033578516], [0, 0, 1, 0], [0, 0, 0, 0], [9E9, 9E9, 9E9, 9E9, 9E9, 9E9]];
    CONST robtarget p4230:= [[1520.8261742525665, -51.54719955056562, 993.500033578516], [0, 0, 1, 0], [0, 0, 0, 0], [9E9, 9E9, 9E9, 9E9, 9E9, 9E9]];
    CONST robtarget p4231:= [[1520.55210150569, -51.650111266866645, 993.500033578516], [0, 0, 1, 0], [0, 0, 0, 0], [9E9, 9E9, 9E9, 9E9, 9E9, 9E9]];
    CONST robtarget p4232:= [[1519.9544210839522, -51.87907929459036, 993.500033578516], [0, 0, 1, 0], [0, 0, 0, 0], [9E9, 9E9, 9E9, 9E9, 9E9, 9E9]];
    CONST robtarget p4233:= [[1519.5517712169235, -52.0190080165721, 993.500033578516], [0, 0, 1, 0], [0, 0, 0, 0], [9E9, 9E9, 9E9, 9E9, 9E9, 9E9]];
    CONST robtarget p4234:= [[1519.2269060775236, -52.15534401518349, 993.500033578516], [0, 0, 1, 0], [0, 0, 0, 0], [9E9, 9E9, 9E9, 9E9, 9E9, 9E9]];
    CONST robtarget p4235:= [[1519.0186794130111, -52.22613680111611, 993.500033578516], [0, 0, 1, 0], [0, 0, 0, 0], [9E9, 9E9, 9E9, 9E9, 9E9, 9E9]];
    CONST robtarget p4236:= [[1518.6179406669776, -52.38998721346795, 993.500033578516], [0, 0, 1, 0], [0, 0, 0, 0], [9E9, 9E9, 9E9, 9E9, 9E9, 9E9]];
    CONST robtarget p4237:= [[1518.4587870960263, -52.446138490118585, 993.500033578516], [0, 0, 1, 0], [0, 0, 0, 0], [9E9, 9E9, 9E9, 9E9, 9E9, 9E9]];
    CONST robtarget p4238:= [[1518.0196676618943, -52.62184867235988, 993.500033578516], [0, 0, 1, 0], [0, 0, 0, 0], [9E9, 9E9, 9E9, 9E9, 9E9, 9E9]];
    CONST robtarget p4239:= [[1517.9462491765103, -52.64270939733751, 993.500033578516], [0, 0, 1, 0], [0, 0, 0, 0], [9E9, 9E9, 9E9, 9E9, 9E9, 9E9]];
    CONST robtarget p4240:= [[1517.8452133160054, -52.66954626238196, 993.500033578516], [0, 0, 1, 0], [0, 0, 0, 0], [9E9, 9E9, 9E9, 9E9, 9E9, 9E9]];
    CONST robtarget p4241:= [[1517.539409203478, -52.755794351686504, 993.500033578516], [0, 0, 1, 0], [0, 0, 0, 0], [9E9, 9E9, 9E9, 9E9, 9E9, 9E9]];
    CONST robtarget p4242:= [[1517.2374200565328, -52.84517201830888, 993.500033578516], [0, 0, 1, 0], [0, 0, 0, 0], [9E9, 9E9, 9E9, 9E9, 9E9, 9E9]];
    CONST robtarget p4243:= [[1516.776050677364, -52.99896724762243, 993.500033578516], [0, 0, 1, 0], [0, 0, 0, 0], [9E9, 9E9, 9E9, 9E9, 9E9, 9E9]];
    CONST robtarget p4244:= [[1516.581299117185, -53.05275866966109, 993.500033578516], [0, 0, 1, 0], [0, 0, 0, 0], [9E9, 9E9, 9E9, 9E9, 9E9, 9E9]];
    CONST robtarget p4245:= [[1516.2463978170776, -53.1566796702992, 993.500033578516], [0, 0, 1, 0], [0, 0, 0, 0], [9E9, 9E9, 9E9, 9E9, 9E9, 9E9]];
    CONST robtarget p4246:= [[1515.897264621398, -53.25665668997287, 993.500033578516], [0, 0, 1, 0], [0, 0, 0, 0], [9E9, 9E9, 9E9, 9E9, 9E9, 9E9]];
    CONST robtarget p4247:= [[1515.7721611934446, -53.294321407000254, 993.500033578516], [0, 0, 1, 0], [0, 0, 0, 0], [9E9, 9E9, 9E9, 9E9, 9E9, 9E9]];
    CONST robtarget p4248:= [[1515.487380039119, -53.37868934300438, 993.500033578516], [0, 0, 1, 0], [0, 0, 0, 0], [9E9, 9E9, 9E9, 9E9, 9E9, 9E9]];
    CONST robtarget p4249:= [[1515.3132971471707, -53.42771482735159, 993.500033578516], [0, 0, 1, 0], [0, 0, 0, 0], [9E9, 9E9, 9E9, 9E9, 9E9, 9E9]];
    CONST robtarget p4250:= [[1515.0162157489547, -53.526027611737376, 993.500033578516], [0, 0, 1, 0], [0, 0, 0, 0], [9E9, 9E9, 9E9, 9E9, 9E9, 9E9]];
    CONST robtarget p4251:= [[1514.8511214577059, -53.574856945271016, 993.500033578516], [0, 0, 1, 0], [0, 0, 0, 0], [9E9, 9E9, 9E9, 9E9, 9E9, 9E9]];
    CONST robtarget p4252:= [[1514.819599401767, -53.582607559393324, 993.500033578516], [0, 0, 1, 0], [0, 0, 0, 0], [9E9, 9E9, 9E9, 9E9, 9E9, 9E9]];
    CONST robtarget p4253:= [[1514.4634535735029, -53.68024438148048, 993.500033578516], [0, 0, 1, 0], [0, 0, 0, 0], [9E9, 9E9, 9E9, 9E9, 9E9, 9E9]];
    CONST robtarget p4254:= [[1514.0493199690436, -53.8190428481932, 993.500033578516], [0, 0, 1, 0], [0, 0, 0, 0], [9E9, 9E9, 9E9, 9E9, 9E9, 9E9]];
    CONST robtarget p4255:= [[1513.782191794132, -53.86996789075499, 993.500033578516], [0, 0, 1, 0], [0, 0, 0, 0], [9E9, 9E9, 9E9, 9E9, 9E9, 9E9]];
    CONST robtarget p4256:= [[1513.3942907577286, -53.9577108957173, 993.500033578516], [0, 0, 1, 0], [0, 0, 0, 0], [9E9, 9E9, 9E9, 9E9, 9E9, 9E9]];
    CONST robtarget p4257:= [[1513.0507526578112, -54.03162418265124, 993.500033578516], [0, 0, 1, 0], [0, 0, 0, 0], [9E9, 9E9, 9E9, 9E9, 9E9, 9E9]];
    CONST robtarget p4258:= [[1512.790702332388, -54.09042850100789, 993.500033578516], [0, 0, 1, 0], [0, 0, 0, 0], [9E9, 9E9, 9E9, 9E9, 9E9, 9E9]];
    CONST robtarget p4259:= [[1512.2345251822828, -54.22341823255052, 993.500033578516], [0, 0, 1, 0], [0, 0, 0, 0], [9E9, 9E9, 9E9, 9E9, 9E9, 9E9]];
    CONST robtarget p4260:= [[1511.7500890319127, -54.327808118398025, 993.500033578516], [0, 0, 1, 0], [0, 0, 0, 0], [9E9, 9E9, 9E9, 9E9, 9E9, 9E9]];
    CONST robtarget p4261:= [[1511.4901620207681, -54.385029805214984, 993.500033578516], [0, 0, 1, 0], [0, 0, 0, 0], [9E9, 9E9, 9E9, 9E9, 9E9, 9E9]];
    CONST robtarget p4262:= [[1511.275113803435, -54.435314142538694, 993.500033578516], [0, 0, 1, 0], [0, 0, 0, 0], [9E9, 9E9, 9E9, 9E9, 9E9, 9E9]];
    CONST robtarget p4263:= [[1511.091027858132, -54.47697870243079, 993.500033578516], [0, 0, 1, 0], [0, 0, 0, 0], [9E9, 9E9, 9E9, 9E9, 9E9, 9E9]];
    CONST robtarget p4264:= [[1510.631634880499, -54.58163304032525, 993.500033578516], [0, 0, 1, 0], [0, 0, 0, 0], [9E9, 9E9, 9E9, 9E9, 9E9, 9E9]];
    CONST robtarget p4265:= [[1509.8866777524872, -54.730203604826464, 993.500033578516], [0, 0, 1, 0], [0, 0, 0, 0], [9E9, 9E9, 9E9, 9E9, 9E9, 9E9]];
    CONST robtarget p4266:= [[1509.5986091573159, -54.76896774149727, 993.500033578516], [0, 0, 1, 0], [0, 0, 0, 0], [9E9, 9E9, 9E9, 9E9, 9E9, 9E9]];
    CONST robtarget p4267:= [[1509.4623916145683, -54.789064651596995, 993.500033578516], [0, 0, 1, 0], [0, 0, 0, 0], [9E9, 9E9, 9E9, 9E9, 9E9, 9E9]];
    CONST robtarget p4268:= [[1509.1727193289246, -54.82535163168283, 993.500033578516], [0, 0, 1, 0], [0, 0, 0, 0], [9E9, 9E9, 9E9, 9E9, 9E9, 9E9]];
    CONST robtarget p4269:= [[1508.8874156709733, -54.87193963453893, 993.500033578516], [0, 0, 1, 0], [0, 0, 0, 0], [9E9, 9E9, 9E9, 9E9, 9E9, 9E9]];
    CONST robtarget p4270:= [[1508.280342828873, -54.96502068016268, 993.500033578516], [0, 0, 1, 0], [0, 0, 0, 0], [9E9, 9E9, 9E9, 9E9, 9E9, 9E9]];
    CONST robtarget p4271:= [[1507.8711718530283, -55.006067498961464, 993.500033578516], [0, 0, 1, 0], [0, 0, 0, 0], [9E9, 9E9, 9E9, 9E9, 9E9, 9E9]];
    CONST robtarget p4272:= [[1507.4012715484357, -55.09119764420451, 993.500033578516], [0, 0, 1, 0], [0, 0, 0, 0], [9E9, 9E9, 9E9, 9E9, 9E9, 9E9]];
    CONST robtarget p4273:= [[1507.1825375348337, -55.111649778817046, 993.500033578516], [0, 0, 1, 0], [0, 0, 0, 0], [9E9, 9E9, 9E9, 9E9, 9E9, 9E9]];
    CONST robtarget p4274:= [[1506.9405789639634, -55.14445017002088, 993.500033578516], [0, 0, 1, 0], [0, 0, 0, 0], [9E9, 9E9, 9E9, 9E9, 9E9, 9E9]];
    CONST robtarget p4275:= [[1506.7951816322957, -55.16475440316749, 993.500033578516], [0, 0, 1, 0], [0, 0, 0, 0], [9E9, 9E9, 9E9, 9E9, 9E9, 9E9]];
    CONST robtarget p4276:= [[1506.4341972707482, -55.23362855509076, 993.500033578516], [0, 0, 1, 0], [0, 0, 0, 0], [9E9, 9E9, 9E9, 9E9, 9E9, 9E9]];
    CONST robtarget p4277:= [[1506.197334481687, -55.27109603195363, 993.500033578516], [0, 0, 1, 0], [0, 0, 0, 0], [9E9, 9E9, 9E9, 9E9, 9E9, 9E9]];
    CONST robtarget p4278:= [[1505.7729826368266, -55.30279009383807, 993.500033578516], [0, 0, 1, 0], [0, 0, 0, 0], [9E9, 9E9, 9E9, 9E9, 9E9, 9E9]];
    CONST robtarget p4279:= [[1505.193360844482, -55.34119761659642, 993.500033578516], [0, 0, 1, 0], [0, 0, 0, 0], [9E9, 9E9, 9E9, 9E9, 9E9, 9E9]];
    CONST robtarget p4280:= [[1505.1091787138334, -55.3518947466569, 993.500033578516], [0, 0, 1, 0], [0, 0, 0, 0], [9E9, 9E9, 9E9, 9E9, 9E9, 9E9]];
    CONST robtarget p4281:= [[1504.623500423256, -55.38234040155617, 993.500033578516], [0, 0, 1, 0], [0, 0, 0, 0], [9E9, 9E9, 9E9, 9E9, 9E9, 9E9]];
    CONST robtarget p4282:= [[1504.2846506156368, -55.40018463009833, 993.500033578516], [0, 0, 1, 0], [0, 0, 0, 0], [9E9, 9E9, 9E9, 9E9, 9E9, 9E9]];
    CONST robtarget p4283:= [[1503.8299638641183, -55.448837768486236, 993.500033578516], [0, 0, 1, 0], [0, 0, 0, 0], [9E9, 9E9, 9E9, 9E9, 9E9, 9E9]];
    CONST robtarget p4284:= [[1503.7590777568064, -55.4582352849862, 993.500033578516], [0, 0, 1, 0], [0, 0, 0, 0], [9E9, 9E9, 9E9, 9E9, 9E9, 9E9]];
    CONST robtarget p4285:= [[1503.1756860825487, -55.50039252686035, 993.500033578516], [0, 0, 1, 0], [0, 0, 0, 0], [9E9, 9E9, 9E9, 9E9, 9E9, 9E9]];
    CONST robtarget p4286:= [[1502.4761824688708, -55.54418570233764, 993.500033578516], [0, 0, 1, 0], [0, 0, 0, 0], [9E9, 9E9, 9E9, 9E9, 9E9, 9E9]];
    CONST robtarget p4287:= [[1502.0740571828355, -55.56668455692807, 993.500033578516], [0, 0, 1, 0], [0, 0, 0, 0], [9E9, 9E9, 9E9, 9E9, 9E9, 9E9]];
    CONST robtarget p4288:= [[1501.7614702870983, -55.576469788016205, 993.500033578516], [0, 0, 1, 0], [0, 0, 0, 0], [9E9, 9E9, 9E9, 9E9, 9E9, 9E9]];
    CONST robtarget p4289:= [[1501.572407141827, -55.587250125592796, 993.500033578516], [0, 0, 1, 0], [0, 0, 0, 0], [9E9, 9E9, 9E9, 9E9, 9E9, 9E9]];
    CONST robtarget p4290:= [[1501.2407053718068, -55.58411707704984, 993.500033578516], [0, 0, 1, 0], [0, 0, 0, 0], [9E9, 9E9, 9E9, 9E9, 9E9, 9E9]];
    CONST robtarget p4291:= [[1500.7502626200526, -55.58631340864275, 993.500033578516], [0, 0, 1, 0], [0, 0, 0, 0], [9E9, 9E9, 9E9, 9E9, 9E9, 9E9]];
    CONST robtarget p4292:= [[1500.076136207753, -55.578782124659185, 993.500033578516], [0, 0, 1, 0], [0, 0, 0, 0], [9E9, 9E9, 9E9, 9E9, 9E9, 9E9]];
    CONST robtarget p4293:= [[1499.8352851728432, -55.58700404388368, 993.500033578516], [0, 0, 1, 0], [0, 0, 0, 0], [9E9, 9E9, 9E9, 9E9, 9E9, 9E9]];
    CONST robtarget p4294:= [[1499.3111495624278, -55.58338391038387, 993.500033578516], [0, 0, 1, 0], [0, 0, 0, 0], [9E9, 9E9, 9E9, 9E9, 9E9, 9E9]];
    CONST robtarget p4295:= [[1498.8450178422254, -55.57016289814243, 993.500033578516], [0, 0, 1, 0], [0, 0, 0, 0], [9E9, 9E9, 9E9, 9E9, 9E9, 9E9]];
    CONST robtarget p4296:= [[1498.5294440360556, -55.576395739153156, 993.500033578516], [0, 0, 1, 0], [0, 0, 0, 0], [9E9, 9E9, 9E9, 9E9, 9E9, 9E9]];
    CONST robtarget p4297:= [[1498.0176023767965, -55.587530262897346, 993.500033578516], [0, 0, 1, 0], [0, 0, 0, 0], [9E9, 9E9, 9E9, 9E9, 9E9, 9E9]];
    CONST robtarget p4298:= [[1497.4225599822685, -55.533677132023925, 993.500033578516], [0, 0, 1, 0], [0, 0, 0, 0], [9E9, 9E9, 9E9, 9E9, 9E9, 9E9]];
    CONST robtarget p4299:= [[1496.957307495406, -55.507272716299724, 993.500033578516], [0, 0, 1, 0], [0, 0, 0, 0], [9E9, 9E9, 9E9, 9E9, 9E9, 9E9]];
    CONST robtarget p4300:= [[1496.4896013300734, -55.47788342910046, 993.500033578516], [0, 0, 1, 0], [0, 0, 0, 0], [9E9, 9E9, 9E9, 9E9, 9E9, 9E9]];
    CONST robtarget p4301:= [[1496.3332440084546, -55.46577199267375, 993.500033578516], [0, 0, 1, 0], [0, 0, 0, 0], [9E9, 9E9, 9E9, 9E9, 9E9, 9E9]];
    CONST robtarget p4302:= [[1496.146425026348, -55.45330333910701, 993.500033578516], [0, 0, 1, 0], [0, 0, 0, 0], [9E9, 9E9, 9E9, 9E9, 9E9, 9E9]];
    CONST robtarget p4303:= [[1495.7627464928887, -55.42756900532496, 993.500033578516], [0, 0, 1, 0], [0, 0, 0, 0], [9E9, 9E9, 9E9, 9E9, 9E9, 9E9]];
    CONST robtarget p4304:= [[1495.5868603620524, -55.41159909679597, 993.500033578516], [0, 0, 1, 0], [0, 0, 0, 0], [9E9, 9E9, 9E9, 9E9, 9E9, 9E9]];
    CONST robtarget p4305:= [[1494.956770261204, -55.353811108585056, 993.500033578516], [0, 0, 1, 0], [0, 0, 0, 0], [9E9, 9E9, 9E9, 9E9, 9E9, 9E9]];
    CONST robtarget p4306:= [[1494.6232404301143, -55.333208732887044, 993.500033578516], [0, 0, 1, 0], [0, 0, 0, 0], [9E9, 9E9, 9E9, 9E9, 9E9, 9E9]];
    CONST robtarget p4307:= [[1494.3824981208945, -55.325648022902456, 993.500033578516], [0, 0, 1, 0], [0, 0, 0, 0], [9E9, 9E9, 9E9, 9E9, 9E9, 9E9]];
    CONST robtarget p4308:= [[1493.9504105921917, -55.282635310347025, 993.500033578516], [0, 0, 1, 0], [0, 0, 0, 0], [9E9, 9E9, 9E9, 9E9, 9E9, 9E9]];
    CONST robtarget p4309:= [[1493.727963888983, -55.25972877084484, 993.500033578516], [0, 0, 1, 0], [0, 0, 0, 0], [9E9, 9E9, 9E9, 9E9, 9E9, 9E9]];
    CONST robtarget p4310:= [[1493.5086219332936, -55.230347852356296, 993.500033578516], [0, 0, 1, 0], [0, 0, 0, 0], [9E9, 9E9, 9E9, 9E9, 9E9, 9E9]];
    CONST robtarget p4311:= [[1493.2976973464006, -55.18842063704244, 993.500033578516], [0, 0, 1, 0], [0, 0, 0, 0], [9E9, 9E9, 9E9, 9E9, 9E9, 9E9]];
    CONST robtarget p4312:= [[1492.7614754009928, -55.11573275181307, 993.500033578516], [0, 0, 1, 0], [0, 0, 0, 0], [9E9, 9E9, 9E9, 9E9, 9E9, 9E9]];
    CONST robtarget p4313:= [[1492.0349530139763, -55.01071776559941, 993.500033578516], [0, 0, 1, 0], [0, 0, 0, 0], [9E9, 9E9, 9E9, 9E9, 9E9, 9E9]];
    CONST robtarget p4314:= [[1491.9104556485145, -54.995467637696635, 993.500033578516], [0, 0, 1, 0], [0, 0, 0, 0], [9E9, 9E9, 9E9, 9E9, 9E9, 9E9]];
    CONST robtarget p4315:= [[1491.365994022553, -54.91480722250425, 993.500033578516], [0, 0, 1, 0], [0, 0, 0, 0], [9E9, 9E9, 9E9, 9E9, 9E9, 9E9]];
    CONST robtarget p4316:= [[1490.8994895127823, -54.843055983383245, 993.500033578516], [0, 0, 1, 0], [0, 0, 0, 0], [9E9, 9E9, 9E9, 9E9, 9E9, 9E9]];
    CONST robtarget p4317:= [[1490.682743188496, -54.812817544047995, 993.500033578516], [0, 0, 1, 0], [0, 0, 0, 0], [9E9, 9E9, 9E9, 9E9, 9E9, 9E9]];
    CONST robtarget p4318:= [[1490.0725343491633, -54.72043536073274, 993.500033578516], [0, 0, 1, 0], [0, 0, 0, 0], [9E9, 9E9, 9E9, 9E9, 9E9, 9E9]];
    CONST robtarget p4319:= [[1489.9214382714708, -54.68659422082041, 993.500033578516], [0, 0, 1, 0], [0, 0, 0, 0], [9E9, 9E9, 9E9, 9E9, 9E9, 9E9]];
    CONST robtarget p4320:= [[1489.6714394241455, -54.640453763794646, 993.500033578516], [0, 0, 1, 0], [0, 0, 0, 0], [9E9, 9E9, 9E9, 9E9, 9E9, 9E9]];
    CONST robtarget p4321:= [[1489.1217172814136, -54.5092227636737, 993.500033578516], [0, 0, 1, 0], [0, 0, 0, 0], [9E9, 9E9, 9E9, 9E9, 9E9, 9E9]];
    CONST robtarget p4322:= [[1488.7596017444519, -54.418506532000436, 993.500033578516], [0, 0, 1, 0], [0, 0, 0, 0], [9E9, 9E9, 9E9, 9E9, 9E9, 9E9]];
    CONST robtarget p4323:= [[1488.3029922018925, -54.333033226777125, 993.500033578516], [0, 0, 1, 0], [0, 0, 0, 0], [9E9, 9E9, 9E9, 9E9, 9E9, 9E9]];
    CONST robtarget p4324:= [[1488.1292831882295, -54.29299971233797, 993.500033578516], [0, 0, 1, 0], [0, 0, 0, 0], [9E9, 9E9, 9E9, 9E9, 9E9, 9E9]];
    CONST robtarget p4325:= [[1487.39797883743, -54.13204040085219, 993.500033578516], [0, 0, 1, 0], [0, 0, 0, 0], [9E9, 9E9, 9E9, 9E9, 9E9, 9E9]];
    CONST robtarget p4326:= [[1487.0692815638577, -54.06800524445507, 993.500033578516], [0, 0, 1, 0], [0, 0, 0, 0], [9E9, 9E9, 9E9, 9E9, 9E9, 9E9]];
    CONST robtarget p4327:= [[1486.9103799502627, -54.03023584936359, 993.500033578516], [0, 0, 1, 0], [0, 0, 0, 0], [9E9, 9E9, 9E9, 9E9, 9E9, 9E9]];
    CONST robtarget p4328:= [[1486.6182098121972, -53.953586224602105, 993.500033578516], [0, 0, 1, 0], [0, 0, 0, 0], [9E9, 9E9, 9E9, 9E9, 9E9, 9E9]];
    CONST robtarget p4329:= [[1486.051886395679, -53.837190438333224, 993.500033578516], [0, 0, 1, 0], [0, 0, 0, 0], [9E9, 9E9, 9E9, 9E9, 9E9, 9E9]];
    CONST robtarget p4330:= [[1485.650379922698, -53.732804484189046, 993.500033578516], [0, 0, 1, 0], [0, 0, 0, 0], [9E9, 9E9, 9E9, 9E9, 9E9, 9E9]];
    CONST robtarget p4331:= [[1485.0257270215172, -53.542501811437035, 993.500033578516], [0, 0, 1, 0], [0, 0, 0, 0], [9E9, 9E9, 9E9, 9E9, 9E9, 9E9]];
    CONST robtarget p4332:= [[1484.6005839463635, -53.39297325238115, 993.500033578516], [0, 0, 1, 0], [0, 0, 0, 0], [9E9, 9E9, 9E9, 9E9, 9E9, 9E9]];
    CONST robtarget p4333:= [[1484.1133895675878, -53.26997823663097, 993.500033578516], [0, 0, 1, 0], [0, 0, 0, 0], [9E9, 9E9, 9E9, 9E9, 9E9, 9E9]];
    CONST robtarget p4334:= [[1483.9939270458583, -53.232246866739864, 993.500033578516], [0, 0, 1, 0], [0, 0, 0, 0], [9E9, 9E9, 9E9, 9E9, 9E9, 9E9]];
    CONST robtarget p4335:= [[1483.5182542714479, -53.09250591094003, 993.500033578516], [0, 0, 1, 0], [0, 0, 0, 0], [9E9, 9E9, 9E9, 9E9, 9E9, 9E9]];
    CONST robtarget p4336:= [[1483.1701215386038, -52.98587141718255, 993.500033578516], [0, 0, 1, 0], [0, 0, 0, 0], [9E9, 9E9, 9E9, 9E9, 9E9, 9E9]];
    CONST robtarget p4337:= [[1482.9411047451688, -52.91681595097207, 993.500033578516], [0, 0, 1, 0], [0, 0, 0, 0], [9E9, 9E9, 9E9, 9E9, 9E9, 9E9]];
    CONST robtarget p4338:= [[1482.6513695181825, -52.825770713120356, 993.500033578516], [0, 0, 1, 0], [0, 0, 0, 0], [9E9, 9E9, 9E9, 9E9, 9E9, 9E9]];
    CONST robtarget p4339:= [[1482.5371334257136, -52.79053611254591, 993.500033578516], [0, 0, 1, 0], [0, 0, 0, 0], [9E9, 9E9, 9E9, 9E9, 9E9, 9E9]];
    CONST robtarget p4340:= [[1482.1167286667298, -52.66034807043669, 993.500033578516], [0, 0, 1, 0], [0, 0, 0, 0], [9E9, 9E9, 9E9, 9E9, 9E9, 9E9]];
    CONST robtarget p4341:= [[1481.845956925924, -52.56396421651416, 993.500033578516], [0, 0, 1, 0], [0, 0, 0, 0], [9E9, 9E9, 9E9, 9E9, 9E9, 9E9]];
    CONST robtarget p4342:= [[1481.678516434214, -52.500512110630424, 993.500033578516], [0, 0, 1, 0], [0, 0, 0, 0], [9E9, 9E9, 9E9, 9E9, 9E9, 9E9]];
    CONST robtarget p4343:= [[1481.3550671261025, -52.379854535104855, 993.500033578516], [0, 0, 1, 0], [0, 0, 0, 0], [9E9, 9E9, 9E9, 9E9, 9E9, 9E9]];
    CONST robtarget p4344:= [[1481.204369425806, -52.32004926681436, 993.500033578516], [0, 0, 1, 0], [0, 0, 0, 0], [9E9, 9E9, 9E9, 9E9, 9E9, 9E9]];
    CONST robtarget p4345:= [[1480.8628409090372, -52.184892066019735, 993.500033578516], [0, 0, 1, 0], [0, 0, 0, 0], [9E9, 9E9, 9E9, 9E9, 9E9, 9E9]];
    CONST robtarget p4346:= [[1480.5867349561524, -52.075438223779386, 993.500033578516], [0, 0, 1, 0], [0, 0, 0, 0], [9E9, 9E9, 9E9, 9E9, 9E9, 9E9]];
    CONST robtarget p4347:= [[1480.3479960740906, -51.98991041644267, 993.500033578516], [0, 0, 1, 0], [0, 0, 0, 0], [9E9, 9E9, 9E9, 9E9, 9E9, 9E9]];
    CONST robtarget p4348:= [[1480.1144084024643, -51.9051531703817, 993.500033578516], [0, 0, 1, 0], [0, 0, 0, 0], [9E9, 9E9, 9E9, 9E9, 9E9, 9E9]];
    CONST robtarget p4349:= [[1479.989167314759, -51.855729042006395, 993.500033578516], [0, 0, 1, 0], [0, 0, 0, 0], [9E9, 9E9, 9E9, 9E9, 9E9, 9E9]];
    CONST robtarget p4350:= [[1479.5711189430117, -51.70193703070361, 993.500033578516], [0, 0, 1, 0], [0, 0, 0, 0], [9E9, 9E9, 9E9, 9E9, 9E9, 9E9]];
    CONST robtarget p4351:= [[1479.447712010906, -51.651171277763666, 993.500033578516], [0, 0, 1, 0], [0, 0, 0, 0], [9E9, 9E9, 9E9, 9E9, 9E9, 9E9]];
    CONST robtarget p4352:= [[1479.2768818082739, -51.58308851321445, 993.500033578516], [0, 0, 1, 0], [0, 0, 0, 0], [9E9, 9E9, 9E9, 9E9, 9E9, 9E9]];
    CONST robtarget p4353:= [[1479.1072501020801, -51.514813261805614, 993.500033578516], [0, 0, 1, 0], [0, 0, 0, 0], [9E9, 9E9, 9E9, 9E9, 9E9, 9E9]];
    CONST robtarget p4354:= [[1478.9312066351868, -51.448137216693326, 993.500033578516], [0, 0, 1, 0], [0, 0, 0, 0], [9E9, 9E9, 9E9, 9E9, 9E9, 9E9]];
    CONST robtarget p4355:= [[1478.663129701284, -51.34851538155688, 993.500033578516], [0, 0, 1, 0], [0, 0, 0, 0], [9E9, 9E9, 9E9, 9E9, 9E9, 9E9]];
    CONST robtarget p4356:= [[1478.5189109755886, -51.293592041661974, 993.500033578516], [0, 0, 1, 0], [0, 0, 0, 0], [9E9, 9E9, 9E9, 9E9, 9E9, 9E9]];
    CONST robtarget p4357:= [[1478.0704800654999, -51.10951071282432, 993.500033578516], [0, 0, 1, 0], [0, 0, 0, 0], [9E9, 9E9, 9E9, 9E9, 9E9, 9E9]];
    CONST robtarget p4358:= [[1477.870674981987, -51.013768564345966, 993.500033578516], [0, 0, 1, 0], [0, 0, 0, 0], [9E9, 9E9, 9E9, 9E9, 9E9, 9E9]];
    CONST robtarget p4359:= [[1477.2920679717724, -50.74493517764239, 993.500033578516], [0, 0, 1, 0], [0, 0, 0, 0], [9E9, 9E9, 9E9, 9E9, 9E9, 9E9]];
    CONST robtarget p4360:= [[1476.8374581820165, -50.5234692697943, 993.500033578516], [0, 0, 1, 0], [0, 0, 0, 0], [9E9, 9E9, 9E9, 9E9, 9E9, 9E9]];
    CONST robtarget p4361:= [[1476.6508657104378, -50.43967452742465, 993.500033578516], [0, 0, 1, 0], [0, 0, 0, 0], [9E9, 9E9, 9E9, 9E9, 9E9, 9E9]];
    CONST robtarget p4362:= [[1476.2004729075525, -50.22755592833073, 993.500033578516], [0, 0, 1, 0], [0, 0, 0, 0], [9E9, 9E9, 9E9, 9E9, 9E9, 9E9]];
    CONST robtarget p4363:= [[1475.9979930314423, -50.144509160115646, 993.500033578516], [0, 0, 1, 0], [0, 0, 0, 0], [9E9, 9E9, 9E9, 9E9, 9E9, 9E9]];
    CONST robtarget p4364:= [[1475.5970406278075, -49.94326641345165, 993.500033578516], [0, 0, 1, 0], [0, 0, 0, 0], [9E9, 9E9, 9E9, 9E9, 9E9, 9E9]];
    CONST robtarget p4365:= [[1475.4000052517188, -49.85319259977679, 993.500033578516], [0, 0, 1, 0], [0, 0, 0, 0], [9E9, 9E9, 9E9, 9E9, 9E9, 9E9]];
    CONST robtarget p4366:= [[1474.8662424457918, -49.61393185504133, 993.500033578516], [0, 0, 1, 0], [0, 0, 0, 0], [9E9, 9E9, 9E9, 9E9, 9E9, 9E9]];
    CONST robtarget p4367:= [[1474.6800299430977, -49.52135509480608, 993.500033578516], [0, 0, 1, 0], [0, 0, 0, 0], [9E9, 9E9, 9E9, 9E9, 9E9, 9E9]];
    CONST robtarget p4368:= [[1474.4855769698784, -49.415769384229165, 993.500033578516], [0, 0, 1, 0], [0, 0, 0, 0], [9E9, 9E9, 9E9, 9E9, 9E9, 9E9]];
    CONST robtarget p4369:= [[1474.0130477885423, -49.15702954035436, 993.500033578516], [0, 0, 1, 0], [0, 0, 0, 0], [9E9, 9E9, 9E9, 9E9, 9E9, 9E9]];
    CONST robtarget p4370:= [[1473.4792387497512, -48.86378570072873, 993.500033578516], [0, 0, 1, 0], [0, 0, 0, 0], [9E9, 9E9, 9E9, 9E9, 9E9, 9E9]];
    CONST robtarget p4371:= [[1472.961074047318, -48.552919336729005, 993.500033578516], [0, 0, 1, 0], [0, 0, 0, 0], [9E9, 9E9, 9E9, 9E9, 9E9, 9E9]];
    CONST robtarget p4372:= [[1472.7592503429184, -48.44633419367906, 993.500033578516], [0, 0, 1, 0], [0, 0, 0, 0], [9E9, 9E9, 9E9, 9E9, 9E9, 9E9]];
    CONST robtarget p4373:= [[1472.2831414225227, -48.18974105664824, 993.500033578516], [0, 0, 1, 0], [0, 0, 0, 0], [9E9, 9E9, 9E9, 9E9, 9E9, 9E9]];
    CONST robtarget p4374:= [[1472.0304155777035, -48.04317838496338, 993.500033578516], [0, 0, 1, 0], [0, 0, 0, 0], [9E9, 9E9, 9E9, 9E9, 9E9, 9E9]];
    CONST robtarget p4375:= [[1471.55541880041, -47.76993041378741, 993.500033578516], [0, 0, 1, 0], [0, 0, 0, 0], [9E9, 9E9, 9E9, 9E9, 9E9, 9E9]];
    CONST robtarget p4376:= [[1471.209550609135, -47.571900426464396, 993.500033578516], [0, 0, 1, 0], [0, 0, 0, 0], [9E9, 9E9, 9E9, 9E9, 9E9, 9E9]];
    CONST robtarget p4377:= [[1471.098494904783, -47.51546884866926, 993.500033578516], [0, 0, 1, 0], [0, 0, 0, 0], [9E9, 9E9, 9E9, 9E9, 9E9, 9E9]];
    CONST robtarget p4378:= [[1470.3733746968999, -47.044348302784044, 993.500033578516], [0, 0, 1, 0], [0, 0, 0, 0], [9E9, 9E9, 9E9, 9E9, 9E9, 9E9]];
    CONST robtarget p4379:= [[1470.1659933792707, -46.9109455788919, 993.500033578516], [0, 0, 1, 0], [0, 0, 0, 0], [9E9, 9E9, 9E9, 9E9, 9E9, 9E9]];
    CONST robtarget p4380:= [[1469.9374612494296, -46.76597114284105, 993.500033578516], [0, 0, 1, 0], [0, 0, 0, 0], [9E9, 9E9, 9E9, 9E9, 9E9, 9E9]];
    CONST robtarget p4381:= [[1469.7899181933042, -46.66870560674455, 993.500033578516], [0, 0, 1, 0], [0, 0, 0, 0], [9E9, 9E9, 9E9, 9E9, 9E9, 9E9]];
    CONST robtarget p4382:= [[1469.4871068677887, -46.467041953247715, 993.500033578516], [0, 0, 1, 0], [0, 0, 0, 0], [9E9, 9E9, 9E9, 9E9, 9E9, 9E9]];
    CONST robtarget p4383:= [[1469.1738707744264, -46.262481534371446, 993.500033578516], [0, 0, 1, 0], [0, 0, 0, 0], [9E9, 9E9, 9E9, 9E9, 9E9, 9E9]];
    CONST robtarget p4384:= [[1468.700717128601, -45.944715795300326, 993.500033578516], [0, 0, 1, 0], [0, 0, 0, 0], [9E9, 9E9, 9E9, 9E9, 9E9, 9E9]];
    CONST robtarget p4385:= [[1468.4591924951314, -45.78501448875601, 993.500033578516], [0, 0, 1, 0], [0, 0, 0, 0], [9E9, 9E9, 9E9, 9E9, 9E9, 9E9]];
    CONST robtarget p4386:= [[1468.3149696989965, -45.68948175517657, 993.500033578516], [0, 0, 1, 0], [0, 0, 0, 0], [9E9, 9E9, 9E9, 9E9, 9E9, 9E9]];
    CONST robtarget p4387:= [[1468.1774206105094, -45.60275736882703, 993.500033578516], [0, 0, 1, 0], [0, 0, 0, 0], [9E9, 9E9, 9E9, 9E9, 9E9, 9E9]];
    CONST robtarget p4388:= [[1467.985052291578, -45.468603763654855, 993.500033578516], [0, 0, 1, 0], [0, 0, 0, 0], [9E9, 9E9, 9E9, 9E9, 9E9, 9E9]];
    CONST robtarget p4389:= [[1467.7428988334166, -45.30540728316862, 993.500033578516], [0, 0, 1, 0], [0, 0, 0, 0], [9E9, 9E9, 9E9, 9E9, 9E9, 9E9]];
    CONST robtarget p4390:= [[1467.6737694319434, -45.2565389795156, 993.500033578516], [0, 0, 1, 0], [0, 0, 0, 0], [9E9, 9E9, 9E9, 9E9, 9E9, 9E9]];
    CONST robtarget p4391:= [[1467.507890112717, -45.13211157786894, 993.500033578516], [0, 0, 1, 0], [0, 0, 0, 0], [9E9, 9E9, 9E9, 9E9, 9E9, 9E9]];
    CONST robtarget p4392:= [[1467.3095894177138, -44.99223451084978, 993.500033578516], [0, 0, 1, 0], [0, 0, 0, 0], [9E9, 9E9, 9E9, 9E9, 9E9, 9E9]];
    CONST robtarget p4393:= [[1466.7156786268927, -44.5325765936165, 993.500033578516], [0, 0, 1, 0], [0, 0, 0, 0], [9E9, 9E9, 9E9, 9E9, 9E9, 9E9]];
    CONST robtarget p4394:= [[1466.1547149252724, -44.07624238892599, 993.500033578516], [0, 0, 1, 0], [0, 0, 0, 0], [9E9, 9E9, 9E9, 9E9, 9E9, 9E9]];
    CONST robtarget p4395:= [[1465.7141887325488, -43.74135329651541, 993.500033578516], [0, 0, 1, 0], [0, 0, 0, 0], [9E9, 9E9, 9E9, 9E9, 9E9, 9E9]];
    CONST robtarget p4396:= [[1465.610149273394, -43.65079948885719, 993.500033578516], [0, 0, 1, 0], [0, 0, 0, 0], [9E9, 9E9, 9E9, 9E9, 9E9, 9E9]];
    CONST robtarget p4397:= [[1465.085996082822, -43.24261168762269, 993.500033578516], [0, 0, 1, 0], [0, 0, 0, 0], [9E9, 9E9, 9E9, 9E9, 9E9, 9E9]];
    CONST robtarget p4398:= [[1464.879677485009, -43.101084782225314, 993.500033578516], [0, 0, 1, 0], [0, 0, 0, 0], [9E9, 9E9, 9E9, 9E9, 9E9, 9E9]];
    CONST robtarget p4399:= [[1464.6482931560172, -42.93721108853465, 993.500033578516], [0, 0, 1, 0], [0, 0, 0, 0], [9E9, 9E9, 9E9, 9E9, 9E9, 9E9]];
    CONST robtarget p4400:= [[1464.5127086217378, -42.83113776330015, 993.500033578516], [0, 0, 1, 0], [0, 0, 0, 0], [9E9, 9E9, 9E9, 9E9, 9E9, 9E9]];
    CONST robtarget p4401:= [[1464.1404188797799, -42.50879872218689, 993.500033578516], [0, 0, 1, 0], [0, 0, 0, 0], [9E9, 9E9, 9E9, 9E9, 9E9, 9E9]];
    CONST robtarget p4402:= [[1464.0202426011485, -42.39431645683997, 993.500033578516], [0, 0, 1, 0], [0, 0, 0, 0], [9E9, 9E9, 9E9, 9E9, 9E9, 9E9]];
    CONST robtarget p4403:= [[1463.5668016688264, -41.9854212622401, 993.500033578516], [0, 0, 1, 0], [0, 0, 0, 0], [9E9, 9E9, 9E9, 9E9, 9E9, 9E9]];
    CONST robtarget p4404:= [[1463.4114721022515, -41.847442934925155, 993.500033578516], [0, 0, 1, 0], [0, 0, 0, 0], [9E9, 9E9, 9E9, 9E9, 9E9, 9E9]];
    CONST robtarget p4405:= [[1463.244665830669, -41.686062504769126, 993.500033578516], [0, 0, 1, 0], [0, 0, 0, 0], [9E9, 9E9, 9E9, 9E9, 9E9, 9E9]];
    CONST robtarget p4406:= [[1462.7290212103142, -41.24215976634145, 993.500033578516], [0, 0, 1, 0], [0, 0, 0, 0], [9E9, 9E9, 9E9, 9E9, 9E9, 9E9]];
    CONST robtarget p4407:= [[1462.4088683101647, -40.93310057637957, 993.500033578516], [0, 0, 1, 0], [0, 0, 0, 0], [9E9, 9E9, 9E9, 9E9, 9E9, 9E9]];
    CONST robtarget p4408:= [[1462.1146736109954, -40.66919762841559, 993.500033578516], [0, 0, 1, 0], [0, 0, 0, 0], [9E9, 9E9, 9E9, 9E9, 9E9, 9E9]];
    CONST robtarget p4409:= [[1461.6986854672423, -40.319706464912926, 993.500033578516], [0, 0, 1, 0], [0, 0, 0, 0], [9E9, 9E9, 9E9, 9E9, 9E9, 9E9]];
    CONST robtarget p4410:= [[1461.665032400178, -40.28777709568253, 993.500033578516], [0, 0, 1, 0], [0, 0, 0, 0], [9E9, 9E9, 9E9, 9E9, 9E9, 9E9]];
    CONST robtarget p4411:= [[1461.3747768032515, -40.013730530715804, 993.500033578516], [0, 0, 1, 0], [0, 0, 0, 0], [9E9, 9E9, 9E9, 9E9, 9E9, 9E9]];
    CONST robtarget p4412:= [[1461.2976350925499, -39.94722761113904, 993.500033578516], [0, 0, 1, 0], [0, 0, 0, 0], [9E9, 9E9, 9E9, 9E9, 9E9, 9E9]];
    CONST robtarget p4413:= [[1461.2348011568927, -39.884487773935845, 993.500033578516], [0, 0, 1, 0], [0, 0, 0, 0], [9E9, 9E9, 9E9, 9E9, 9E9, 9E9]];
    CONST robtarget p4414:= [[1461.1414080838474, -39.78724175052098, 993.500033578516], [0, 0, 1, 0], [0, 0, 0, 0], [9E9, 9E9, 9E9, 9E9, 9E9, 9E9]];
    CONST robtarget p4415:= [[1461.0285793417422, -39.67063676383306, 993.500033578516], [0, 0, 1, 0], [0, 0, 0, 0], [9E9, 9E9, 9E9, 9E9, 9E9, 9E9]];
    CONST robtarget p4416:= [[1460.7106398439648, -39.340902137409245, 993.500033578516], [0, 0, 1, 0], [0, 0, 0, 0], [9E9, 9E9, 9E9, 9E9, 9E9, 9E9]];
    CONST robtarget p4417:= [[1460.5259848645633, -39.14810544286311, 993.500033578516], [0, 0, 1, 0], [0, 0, 0, 0], [9E9, 9E9, 9E9, 9E9, 9E9, 9E9]];
    CONST robtarget p4418:= [[1460.3213780341266, -38.923339295912825, 993.500033578516], [0, 0, 1, 0], [0, 0, 0, 0], [9E9, 9E9, 9E9, 9E9, 9E9, 9E9]];
    CONST robtarget p4419:= [[1460.075777415675, -38.678019821477235, 993.500033578516], [0, 0, 1, 0], [0, 0, 0, 0], [9E9, 9E9, 9E9, 9E9, 9E9, 9E9]];
    CONST robtarget p4420:= [[1459.5229982810656, -38.10178260853324, 993.500033578516], [0, 0, 1, 0], [0, 0, 0, 0], [9E9, 9E9, 9E9, 9E9, 9E9, 9E9]];
    CONST robtarget p4421:= [[1459.3173092489187, -37.88251401324446, 993.500033578516], [0, 0, 1, 0], [0, 0, 0, 0], [9E9, 9E9, 9E9, 9E9, 9E9, 9E9]];
    CONST robtarget p4422:= [[1458.9568903150384, -37.52321421058282, 993.500033578516], [0, 0, 1, 0], [0, 0, 0, 0], [9E9, 9E9, 9E9, 9E9, 9E9, 9E9]];
    CONST robtarget p4423:= [[1458.8422749042777, -37.39715324194863, 993.500033578516], [0, 0, 1, 0], [0, 0, 0, 0], [9E9, 9E9, 9E9, 9E9, 9E9, 9E9]];
    CONST robtarget p4424:= [[1458.7430137493998, -37.284780410753285, 993.500033578516], [0, 0, 1, 0], [0, 0, 0, 0], [9E9, 9E9, 9E9, 9E9, 9E9, 9E9]];
    CONST robtarget p4425:= [[1458.4895517709979, -37.01070459612066, 993.500033578516], [0, 0, 1, 0], [0, 0, 0, 0], [9E9, 9E9, 9E9, 9E9, 9E9, 9E9]];
    CONST robtarget p4426:= [[1458.3812173973065, -36.87566878309118, 993.500033578516], [0, 0, 1, 0], [0, 0, 0, 0], [9E9, 9E9, 9E9, 9E9, 9E9, 9E9]];
    CONST robtarget p4427:= [[1458.1143073150267, -36.54860816081012, 993.500033578516], [0, 0, 1, 0], [0, 0, 0, 0], [9E9, 9E9, 9E9, 9E9, 9E9, 9E9]];
    CONST robtarget p4428:= [[1457.8927407616766, -36.30478165148204, 993.500033578516], [0, 0, 1, 0], [0, 0, 0, 0], [9E9, 9E9, 9E9, 9E9, 9E9, 9E9]];
    CONST robtarget p4429:= [[1457.8454890317525, -36.253773133005964, 993.500033578516], [0, 0, 1, 0], [0, 0, 0, 0], [9E9, 9E9, 9E9, 9E9, 9E9, 9E9]];
    CONST robtarget p4430:= [[1457.6680091020612, -36.028133270333846, 993.500033578516], [0, 0, 1, 0], [0, 0, 0, 0], [9E9, 9E9, 9E9, 9E9, 9E9, 9E9]];
    CONST robtarget p4431:= [[1457.5712639042347, -35.90274196024533, 993.500033578516], [0, 0, 1, 0], [0, 0, 0, 0], [9E9, 9E9, 9E9, 9E9, 9E9, 9E9]];
    CONST robtarget p4432:= [[1457.545801344033, -35.87005476594986, 993.500033578516], [0, 0, 1, 0], [0, 0, 0, 0], [9E9, 9E9, 9E9, 9E9, 9E9, 9E9]];
    CONST robtarget p4433:= [[1457.0997122684437, -35.356358318288216, 993.500033578516], [0, 0, 1, 0], [0, 0, 0, 0], [9E9, 9E9, 9E9, 9E9, 9E9, 9E9]];
    CONST robtarget p4434:= [[1456.9196996114706, -35.12680782836004, 993.500033578516], [0, 0, 1, 0], [0, 0, 0, 0], [9E9, 9E9, 9E9, 9E9, 9E9, 9E9]];
    CONST robtarget p4435:= [[1456.5171419510377, -34.64983802862872, 993.500033578516], [0, 0, 1, 0], [0, 0, 0, 0], [9E9, 9E9, 9E9, 9E9, 9E9, 9E9]];
    CONST robtarget p4436:= [[1456.2501829153084, -34.31923470079157, 993.500033578516], [0, 0, 1, 0], [0, 0, 0, 0], [9E9, 9E9, 9E9, 9E9, 9E9, 9E9]];
    CONST robtarget p4437:= [[1456.111690408953, -34.15746797368403, 993.500033578516], [0, 0, 1, 0], [0, 0, 0, 0], [9E9, 9E9, 9E9, 9E9, 9E9, 9E9]];
    CONST robtarget p4438:= [[1455.930833303019, -33.94299949791176, 993.500033578516], [0, 0, 1, 0], [0, 0, 0, 0], [9E9, 9E9, 9E9, 9E9, 9E9, 9E9]];
    CONST robtarget p4439:= [[1455.676524131721, -33.58519866088049, 993.500033578516], [0, 0, 1, 0], [0, 0, 0, 0], [9E9, 9E9, 9E9, 9E9, 9E9, 9E9]];
    CONST robtarget p4440:= [[1455.5382593071217, -33.39332764403457, 993.500033578516], [0, 0, 1, 0], [0, 0, 0, 0], [9E9, 9E9, 9E9, 9E9, 9E9, 9E9]];
    CONST robtarget p4441:= [[1455.3774547792264, -33.17080595346653, 993.500033578516], [0, 0, 1, 0], [0, 0, 0, 0], [9E9, 9E9, 9E9, 9E9, 9E9, 9E9]];
    CONST robtarget p4442:= [[1455.136813000254, -32.82445309837537, 993.500033578516], [0, 0, 1, 0], [0, 0, 0, 0], [9E9, 9E9, 9E9, 9E9, 9E9, 9E9]];
    CONST robtarget p4443:= [[1454.6105241742032, -32.08254331011296, 993.500033578516], [0, 0, 1, 0], [0, 0, 0, 0], [9E9, 9E9, 9E9, 9E9, 9E9, 9E9]];
    CONST robtarget p4444:= [[1454.3300729965454, -31.690579023710512, 993.500033578516], [0, 0, 1, 0], [0, 0, 0, 0], [9E9, 9E9, 9E9, 9E9, 9E9, 9E9]];
    CONST robtarget p4445:= [[1454.2929204864433, -31.643922271611267, 993.500033578516], [0, 0, 1, 0], [0, 0, 0, 0], [9E9, 9E9, 9E9, 9E9, 9E9, 9E9]];
    CONST robtarget p4446:= [[1454.1143006359985, -31.382654989880685, 993.500033578516], [0, 0, 1, 0], [0, 0, 0, 0], [9E9, 9E9, 9E9, 9E9, 9E9, 9E9]];
    CONST robtarget p4447:= [[1453.822769449252, -30.978440321798878, 993.500033578516], [0, 0, 1, 0], [0, 0, 0, 0], [9E9, 9E9, 9E9, 9E9, 9E9, 9E9]];
    CONST robtarget p4448:= [[1453.7956024162304, -30.943963169675783, 993.500033578516], [0, 0, 1, 0], [0, 0, 0, 0], [9E9, 9E9, 9E9, 9E9, 9E9, 9E9]];
    CONST robtarget p4449:= [[1453.4712760211025, -30.47335516310359, 993.500033578516], [0, 0, 1, 0], [0, 0, 0, 0], [9E9, 9E9, 9E9, 9E9, 9E9, 9E9]];
    CONST robtarget p4450:= [[1453.2091838332376, -30.03319082974599, 993.500033578516], [0, 0, 1, 0], [0, 0, 0, 0], [9E9, 9E9, 9E9, 9E9, 9E9, 9E9]];
    CONST robtarget p4451:= [[1452.81482675115, -29.39539609433306, 993.500033578516], [0, 0, 1, 0], [0, 0, 0, 0], [9E9, 9E9, 9E9, 9E9, 9E9, 9E9]];
    CONST robtarget p4452:= [[1452.6626674242139, -29.127003002081096, 993.500033578516], [0, 0, 1, 0], [0, 0, 0, 0], [9E9, 9E9, 9E9, 9E9, 9E9, 9E9]];
    CONST robtarget p4453:= [[1452.4509852010776, -28.783090172232797, 993.500033578516], [0, 0, 1, 0], [0, 0, 0, 0], [9E9, 9E9, 9E9, 9E9, 9E9, 9E9]];
    CONST robtarget p4454:= [[1452.2716586626552, -28.494094816402367, 993.500033578516], [0, 0, 1, 0], [0, 0, 0, 0], [9E9, 9E9, 9E9, 9E9, 9E9, 9E9]];
    CONST robtarget p4455:= [[1452.1760655094763, -28.33280689550005, 993.500033578516], [0, 0, 1, 0], [0, 0, 0, 0], [9E9, 9E9, 9E9, 9E9, 9E9, 9E9]];
    CONST robtarget p4456:= [[1452.0184667117157, -28.092057127832007, 993.500033578516], [0, 0, 1, 0], [0, 0, 0, 0], [9E9, 9E9, 9E9, 9E9, 9E9, 9E9]];
    CONST robtarget p4457:= [[1451.889574507297, -27.865251420437474, 993.500033578516], [0, 0, 1, 0], [0, 0, 0, 0], [9E9, 9E9, 9E9, 9E9, 9E9, 9E9]];
    CONST robtarget p4458:= [[1451.7593452706672, -27.645309795740587, 993.500033578516], [0, 0, 1, 0], [0, 0, 0, 0], [9E9, 9E9, 9E9, 9E9, 9E9, 9E9]];
    CONST robtarget p4459:= [[1451.5810118163602, -27.347003420867622, 993.500033578516], [0, 0, 1, 0], [0, 0, 0, 0], [9E9, 9E9, 9E9, 9E9, 9E9, 9E9]];
    CONST robtarget p4460:= [[1451.415405754412, -27.08044512164929, 993.500033578516], [0, 0, 1, 0], [0, 0, 0, 0], [9E9, 9E9, 9E9, 9E9, 9E9, 9E9]];
    CONST robtarget p4461:= [[1451.323510736806, -26.894246207522514, 993.500033578516], [0, 0, 1, 0], [0, 0, 0, 0], [9E9, 9E9, 9E9, 9E9, 9E9, 9E9]];
    CONST robtarget p4462:= [[1451.1778371421158, -26.60611060888759, 993.500033578516], [0, 0, 1, 0], [0, 0, 0, 0], [9E9, 9E9, 9E9, 9E9, 9E9, 9E9]];
    CONST robtarget p4463:= [[1450.978139912826, -26.191976259445482, 993.500033578516], [0, 0, 1, 0], [0, 0, 0, 0], [9E9, 9E9, 9E9, 9E9, 9E9, 9E9]];
    CONST robtarget p4464:= [[1450.8874136799914, -26.00984996607812, 993.500033578516], [0, 0, 1, 0], [0, 0, 0, 0], [9E9, 9E9, 9E9, 9E9, 9E9, 9E9]];
    CONST robtarget p4465:= [[1450.6495442113712, -25.594648699731138, 993.500033578516], [0, 0, 1, 0], [0, 0, 0, 0], [9E9, 9E9, 9E9, 9E9, 9E9, 9E9]];
    CONST robtarget p4466:= [[1450.5022522014378, -25.289847648122297, 993.500033578516], [0, 0, 1, 0], [0, 0, 0, 0], [9E9, 9E9, 9E9, 9E9, 9E9, 9E9]];
    CONST robtarget p4467:= [[1450.4130950225212, -25.114675434013286, 993.500033578516], [0, 0, 1, 0], [0, 0, 0, 0], [9E9, 9E9, 9E9, 9E9, 9E9, 9E9]];
    CONST robtarget p4468:= [[1450.3436790401875, -24.9765874454923, 993.500033578516], [0, 0, 1, 0], [0, 0, 0, 0], [9E9, 9E9, 9E9, 9E9, 9E9, 9E9]];
    CONST robtarget p4469:= [[1450.152343869645, -24.61668945609481, 993.500033578516], [0, 0, 1, 0], [0, 0, 0, 0], [9E9, 9E9, 9E9, 9E9, 9E9, 9E9]];
    CONST robtarget p4470:= [[1450.093339734578, -24.502238099036667, 993.500033578516], [0, 0, 1, 0], [0, 0, 0, 0], [9E9, 9E9, 9E9, 9E9, 9E9, 9E9]];
    CONST robtarget p4471:= [[1449.8858297453678, -24.093244705000032, 993.500033578516], [0, 0, 1, 0], [0, 0, 0, 0], [9E9, 9E9, 9E9, 9E9, 9E9, 9E9]];
    CONST robtarget p4472:= [[1449.601651616766, -23.51723585393284, 993.500033578516], [0, 0, 1, 0], [0, 0, 0, 0], [9E9, 9E9, 9E9, 9E9, 9E9, 9E9]];
    CONST robtarget p4473:= [[1449.4184228187078, -23.091352777064955, 993.500033578516], [0, 0, 1, 0], [0, 0, 0, 0], [9E9, 9E9, 9E9, 9E9, 9E9, 9E9]];
    CONST robtarget p4474:= [[1449.257760634686, -22.728243642610266, 993.500033578516], [0, 0, 1, 0], [0, 0, 0, 0], [9E9, 9E9, 9E9, 9E9, 9E9, 9E9]];
    CONST robtarget p4475:= [[1449.1097620808712, -22.377918104530224, 993.500033578516], [0, 0, 1, 0], [0, 0, 0, 0], [9E9, 9E9, 9E9, 9E9, 9E9, 9E9]];
    CONST robtarget p4476:= [[1448.904544979288, -21.867866621248076, 993.500033578516], [0, 0, 1, 0], [0, 0, 0, 0], [9E9, 9E9, 9E9, 9E9, 9E9, 9E9]];
    CONST robtarget p4477:= [[1448.787147048693, -21.60081505089618, 993.500033578516], [0, 0, 1, 0], [0, 0, 0, 0], [9E9, 9E9, 9E9, 9E9, 9E9, 9E9]];
    CONST robtarget p4478:= [[1448.4803760566238, -20.86852765070652, 993.500033578516], [0, 0, 1, 0], [0, 0, 0, 0], [9E9, 9E9, 9E9, 9E9, 9E9, 9E9]];
    CONST robtarget p4479:= [[1448.219025891624, -20.262632641558, 993.500033578516], [0, 0, 1, 0], [0, 0, 0, 0], [9E9, 9E9, 9E9, 9E9, 9E9, 9E9]];
    CONST robtarget p4480:= [[1448.028353344372, -19.776100207575695, 993.500033578516], [0, 0, 1, 0], [0, 0, 0, 0], [9E9, 9E9, 9E9, 9E9, 9E9, 9E9]];
    CONST robtarget p4481:= [[1447.9662801234595, -19.60038009290072, 993.500033578516], [0, 0, 1, 0], [0, 0, 0, 0], [9E9, 9E9, 9E9, 9E9, 9E9, 9E9]];
    CONST robtarget p4482:= [[1447.883716032291, -19.393439845961694, 993.500033578516], [0, 0, 1, 0], [0, 0, 0, 0], [9E9, 9E9, 9E9, 9E9, 9E9, 9E9]];
    CONST robtarget p4483:= [[1447.7651239481486, -19.04817060263818, 993.500033578516], [0, 0, 1, 0], [0, 0, 0, 0], [9E9, 9E9, 9E9, 9E9, 9E9, 9E9]];
    CONST robtarget p4484:= [[1447.7437592759402, -18.97900298494855, 993.500033578516], [0, 0, 1, 0], [0, 0, 0, 0], [9E9, 9E9, 9E9, 9E9, 9E9, 9E9]];
    CONST robtarget p4485:= [[1447.5319696866477, -18.371255655215563, 993.500033578516], [0, 0, 1, 0], [0, 0, 0, 0], [9E9, 9E9, 9E9, 9E9, 9E9, 9E9]];
    CONST robtarget p4486:= [[1447.448269507716, -18.073888614757784, 993.500033578516], [0, 0, 1, 0], [0, 0, 0, 0], [9E9, 9E9, 9E9, 9E9, 9E9, 9E9]];
    CONST robtarget p4487:= [[1447.2825869151648, -17.606555345175202, 993.500033578516], [0, 0, 1, 0], [0, 0, 0, 0], [9E9, 9E9, 9E9, 9E9, 9E9, 9E9]];
    CONST robtarget p4488:= [[1447.2489928620935, -17.521057426415233, 993.500033578516], [0, 0, 1, 0], [0, 0, 0, 0], [9E9, 9E9, 9E9, 9E9, 9E9, 9E9]];
    CONST robtarget p4489:= [[1447.100496593344, -17.119656366294727, 993.500033578516], [0, 0, 1, 0], [0, 0, 0, 0], [9E9, 9E9, 9E9, 9E9, 9E9, 9E9]];
    CONST robtarget p4490:= [[1446.8399638672424, -16.318046393287624, 993.500033578516], [0, 0, 1, 0], [0, 0, 0, 0], [9E9, 9E9, 9E9, 9E9, 9E9, 9E9]];
    CONST robtarget p4491:= [[1446.6117105513147, -15.527764181139169, 993.500033578516], [0, 0, 1, 0], [0, 0, 0, 0], [9E9, 9E9, 9E9, 9E9, 9E9, 9E9]];
    CONST robtarget p4492:= [[1446.5908206679558, -15.457181947789365, 993.500033578516], [0, 0, 1, 0], [0, 0, 0, 0], [9E9, 9E9, 9E9, 9E9, 9E9, 9E9]];
    CONST robtarget p4493:= [[1446.557513808863, -15.325228575060883, 993.500033578516], [0, 0, 1, 0], [0, 0, 0, 0], [9E9, 9E9, 9E9, 9E9, 9E9, 9E9]];
    CONST robtarget p4494:= [[1446.445181637588, -14.892041010785022, 993.500033578516], [0, 0, 1, 0], [0, 0, 0, 0], [9E9, 9E9, 9E9, 9E9, 9E9, 9E9]];
    CONST robtarget p4495:= [[1446.3638744086088, -14.623622527065073, 993.500033578516], [0, 0, 1, 0], [0, 0, 0, 0], [9E9, 9E9, 9E9, 9E9, 9E9, 9E9]];
    CONST robtarget p4496:= [[1446.248695598827, -14.192144901246913, 993.500033578516], [0, 0, 1, 0], [0, 0, 0, 0], [9E9, 9E9, 9E9, 9E9, 9E9, 9E9]];
    CONST robtarget p4497:= [[1446.2130586447283, -14.042024428792807, 993.500033578516], [0, 0, 1, 0], [0, 0, 0, 0], [9E9, 9E9, 9E9, 9E9, 9E9, 9E9]];
    CONST robtarget p4498:= [[1446.1801863346998, -13.900479650548888, 993.500033578516], [0, 0, 1, 0], [0, 0, 0, 0], [9E9, 9E9, 9E9, 9E9, 9E9, 9E9]];
    CONST robtarget p4499:= [[1446.1379006529303, -13.73809601356546, 993.500033578516], [0, 0, 1, 0], [0, 0, 0, 0], [9E9, 9E9, 9E9, 9E9, 9E9, 9E9]];
    CONST robtarget p4500:= [[1446.0898901205442, -13.52617807656128, 993.500033578516], [0, 0, 1, 0], [0, 0, 0, 0], [9E9, 9E9, 9E9, 9E9, 9E9, 9E9]];
    CONST robtarget p4501:= [[1445.96869204235, -13.084649917623992, 993.500033578516], [0, 0, 1, 0], [0, 0, 0, 0], [9E9, 9E9, 9E9, 9E9, 9E9, 9E9]];
    CONST robtarget p4502:= [[1445.880459516816, -12.71206127059478, 993.500033578516], [0, 0, 1, 0], [0, 0, 0, 0], [9E9, 9E9, 9E9, 9E9, 9E9, 9E9]];
    CONST robtarget p4503:= [[1445.8444928383797, -12.575779129445642, 993.500033578516], [0, 0, 1, 0], [0, 0, 0, 0], [9E9, 9E9, 9E9, 9E9, 9E9, 9E9]];
    CONST robtarget p4504:= [[1445.7687421230473, -12.295723847219456, 993.500033578516], [0, 0, 1, 0], [0, 0, 0, 0], [9E9, 9E9, 9E9, 9E9, 9E9, 9E9]];
    CONST robtarget p4505:= [[1445.7434997946361, -12.190437467055787, 993.500033578516], [0, 0, 1, 0], [0, 0, 0, 0], [9E9, 9E9, 9E9, 9E9, 9E9, 9E9]];
    CONST robtarget p4506:= [[1445.6696976260655, -11.906670603858409, 993.500033578516], [0, 0, 1, 0], [0, 0, 0, 0], [9E9, 9E9, 9E9, 9E9, 9E9, 9E9]];
    CONST robtarget p4507:= [[1445.6361381338247, -11.737292993238505, 993.500033578516], [0, 0, 1, 0], [0, 0, 0, 0], [9E9, 9E9, 9E9, 9E9, 9E9, 9E9]];
    CONST robtarget p4508:= [[1445.5686237899918, -11.376670982411127, 993.500033578516], [0, 0, 1, 0], [0, 0, 0, 0], [9E9, 9E9, 9E9, 9E9, 9E9, 9E9]];
    CONST robtarget p4509:= [[1445.505837607022, -10.955177036231255, 993.500033578516], [0, 0, 1, 0], [0, 0, 0, 0], [9E9, 9E9, 9E9, 9E9, 9E9, 9E9]];
    CONST robtarget p4510:= [[1445.409306350668, -10.343968819645049, 993.500033578516], [0, 0, 1, 0], [0, 0, 0, 0], [9E9, 9E9, 9E9, 9E9, 9E9, 9E9]];
    CONST robtarget p4511:= [[1445.2724718050704, -9.758343678615404, 993.500033578516], [0, 0, 1, 0], [0, 0, 0, 0], [9E9, 9E9, 9E9, 9E9, 9E9, 9E9]];
    CONST robtarget p4512:= [[1445.2143581407472, -9.379810719556517, 993.500033578516], [0, 0, 1, 0], [0, 0, 0, 0], [9E9, 9E9, 9E9, 9E9, 9E9, 9E9]];
    CONST robtarget p4513:= [[1445.1859734945415, -9.21441551167485, 993.500033578516], [0, 0, 1, 0], [0, 0, 0, 0], [9E9, 9E9, 9E9, 9E9, 9E9, 9E9]];
    CONST robtarget p4514:= [[1445.0402287695113, -8.525664131560966, 993.500033578516], [0, 0, 1, 0], [0, 0, 0, 0], [9E9, 9E9, 9E9, 9E9, 9E9, 9E9]];
    CONST robtarget p4515:= [[1444.9673793536524, -8.09909476667604, 993.500033578516], [0, 0, 1, 0], [0, 0, 0, 0], [9E9, 9E9, 9E9, 9E9, 9E9, 9E9]];
    CONST robtarget p4516:= [[1444.9392274804798, -7.828558934190603, 993.500033578516], [0, 0, 1, 0], [0, 0, 0, 0], [9E9, 9E9, 9E9, 9E9, 9E9, 9E9]];
    CONST robtarget p4517:= [[1444.934363656754, -7.789613861520294, 993.500033578516], [0, 0, 1, 0], [0, 0, 0, 0], [9E9, 9E9, 9E9, 9E9, 9E9, 9E9]];
    CONST robtarget p4518:= [[1444.9078976057003, -7.541704045526274, 993.500033578516], [0, 0, 1, 0], [0, 0, 0, 0], [9E9, 9E9, 9E9, 9E9, 9E9, 9E9]];
    CONST robtarget p4519:= [[1444.8850231470844, -7.279024119913245, 993.500033578516], [0, 0, 1, 0], [0, 0, 0, 0], [9E9, 9E9, 9E9, 9E9, 9E9, 9E9]];
    CONST robtarget p4520:= [[1444.828062279042, -6.879693388657444, 993.500033578516], [0, 0, 1, 0], [0, 0, 0, 0], [9E9, 9E9, 9E9, 9E9, 9E9, 9E9]];
    CONST robtarget p4521:= [[1444.7900644308654, -6.395726105106036, 993.500033578516], [0, 0, 1, 0], [0, 0, 0, 0], [9E9, 9E9, 9E9, 9E9, 9E9, 9E9]];
    CONST robtarget p4522:= [[1444.7342062961845, -5.9127044767689085, 993.500033578516], [0, 0, 1, 0], [0, 0, 0, 0], [9E9, 9E9, 9E9, 9E9, 9E9, 9E9]];
    CONST robtarget p4523:= [[1444.6621485334556, -5.366721876334864, 993.500033578516], [0, 0, 1, 0], [0, 0, 0, 0], [9E9, 9E9, 9E9, 9E9, 9E9, 9E9]];
    CONST robtarget p4524:= [[1444.6122564198968, -4.704455812737365, 993.500033578516], [0, 0, 1, 0], [0, 0, 0, 0], [9E9, 9E9, 9E9, 9E9, 9E9, 9E9]];
    CONST robtarget p4525:= [[1444.5726017023749, -4.333920325690144, 993.500033578516], [0, 0, 1, 0], [0, 0, 0, 0], [9E9, 9E9, 9E9, 9E9, 9E9, 9E9]];
    CONST robtarget p4526:= [[1444.5313205259208, -4.072334927152355, 993.500033578516], [0, 0, 1, 0], [0, 0, 0, 0], [9E9, 9E9, 9E9, 9E9, 9E9, 9E9]];
    CONST robtarget p4527:= [[1444.5212467522767, -3.9912054222854465, 993.500033578516], [0, 0, 1, 0], [0, 0, 0, 0], [9E9, 9E9, 9E9, 9E9, 9E9, 9E9]];
    CONST robtarget p4528:= [[1444.5142758695786, -3.675109895883452, 993.500033578516], [0, 0, 1, 0], [0, 0, 0, 0], [9E9, 9E9, 9E9, 9E9, 9E9, 9E9]];
    CONST robtarget p4529:= [[1444.4929198500688, -3.162645414603446, 993.500033578516], [0, 0, 1, 0], [0, 0, 0, 0], [9E9, 9E9, 9E9, 9E9, 9E9, 9E9]];
    CONST robtarget p4530:= [[1444.4663405446136, -2.5286384905235195, 993.500033578516], [0, 0, 1, 0], [0, 0, 0, 0], [9E9, 9E9, 9E9, 9E9, 9E9, 9E9]];
    CONST robtarget p4531:= [[1444.195236825971, -1.6348780846838622, 994.500033578516], [0, 0, 1, 0], [0, 0, 0, 0], [9E9, 9E9, 9E9, 9E9, 9E9, 9E9]];
    CONST robtarget p4532:= [[1444.1880297553894, -1.4732515699787143, 994.500033578516], [0, 0, 1, 0], [0, 0, 0, 0], [9E9, 9E9, 9E9, 9E9, 9E9, 9E9]];
    CONST robtarget p4533:= [[1444.1833861380526, -1.3156993488799031, 994.500033578516], [0, 0, 1, 0], [0, 0, 0, 0], [9E9, 9E9, 9E9, 9E9, 9E9, 9E9]];
    CONST robtarget p4534:= [[1444.159343230968, -0.7143455506919594, 994.500033578516], [0, 0, 1, 0], [0, 0, 0, 0], [9E9, 9E9, 9E9, 9E9, 9E9, 9E9]];
    CONST robtarget p4535:= [[1444.1450369798067, -0.3134371467546657, 994.500033578516], [0, 0, 1, 0], [0, 0, 0, 0], [9E9, 9E9, 9E9, 9E9, 9E9, 9E9]];
    CONST robtarget p4536:= [[1444.1448337749835, -0.03982398056714942, 994.500033578516], [0, 0, 1, 0], [0, 0, 0, 0], [9E9, 9E9, 9E9, 9E9, 9E9, 9E9]];
    CONST robtarget p4537:= [[1444.1439778939452, 0.29017629654323684, 994.500033578516], [0, 0, 1, 0], [0, 0, 0, 0], [9E9, 9E9, 9E9, 9E9, 9E9, 9E9]];
    CONST robtarget p4538:= [[1444.1549602383368, 0.48887194457519456, 994.500033578516], [0, 0, 1, 0], [0, 0, 0, 0], [9E9, 9E9, 9E9, 9E9, 9E9, 9E9]];
    CONST robtarget p4539:= [[1444.159298181986, 0.5858684512870838, 994.500033578516], [0, 0, 1, 0], [0, 0, 0, 0], [9E9, 9E9, 9E9, 9E9, 9E9, 9E9]];
    CONST robtarget p4540:= [[1444.1682958917972, 0.8179893811821302, 994.500033578516], [0, 0, 1, 0], [0, 0, 0, 0], [9E9, 9E9, 9E9, 9E9, 9E9, 9E9]];
    CONST robtarget p4541:= [[1444.1695381886896, 0.9284446448619548, 994.500033578516], [0, 0, 1, 0], [0, 0, 0, 0], [9E9, 9E9, 9E9, 9E9, 9E9, 9E9]];
    CONST robtarget p4542:= [[1444.2031438447486, 1.5148195606748232, 994.500033578516], [0, 0, 1, 0], [0, 0, 0, 0], [9E9, 9E9, 9E9, 9E9, 9E9, 9E9]];
    CONST robtarget p4543:= [[1444.2105713822853, 2.0332193325005647, 994.500033578516], [0, 0, 1, 0], [0, 0, 0, 0], [9E9, 9E9, 9E9, 9E9, 9E9, 9E9]];
    CONST robtarget p4544:= [[1444.2431133306327, 2.654604892365853, 994.500033578516], [0, 0, 1, 0], [0, 0, 0, 0], [9E9, 9E9, 9E9, 9E9, 9E9, 9E9]];
    CONST robtarget p4545:= [[1444.2445852285002, 2.8196029597429373, 994.500033578516], [0, 0, 1, 0], [0, 0, 0, 0], [9E9, 9E9, 9E9, 9E9, 9E9, 9E9]];
    CONST robtarget p4546:= [[1444.2464722229952, 3.0071636345976174, 994.500033578516], [0, 0, 1, 0], [0, 0, 0, 0], [9E9, 9E9, 9E9, 9E9, 9E9, 9E9]];
    CONST robtarget p4547:= [[1444.2535367748012, 3.300737308137286, 994.500033578516], [0, 0, 1, 0], [0, 0, 0, 0], [9E9, 9E9, 9E9, 9E9, 9E9, 9E9]];
    CONST robtarget p4548:= [[1444.2762002721036, 3.71958380517313, 994.500033578516], [0, 0, 1, 0], [0, 0, 0, 0], [9E9, 9E9, 9E9, 9E9, 9E9, 9E9]];
    CONST robtarget p4549:= [[1444.2927701652313, 4.132844079296163, 994.500033578516], [0, 0, 1, 0], [0, 0, 0, 0], [9E9, 9E9, 9E9, 9E9, 9E9, 9E9]];
    CONST robtarget p4550:= [[1444.30482796831, 4.199267479047279, 994.500033578516], [0, 0, 1, 0], [0, 0, 0, 0], [9E9, 9E9, 9E9, 9E9, 9E9, 9E9]];
    CONST robtarget p4551:= [[1444.3611542389929, 4.574210485856412, 994.500033578516], [0, 0, 1, 0], [0, 0, 0, 0], [9E9, 9E9, 9E9, 9E9, 9E9, 9E9]];
    CONST robtarget p4552:= [[1444.398661693175, 5.052341444579838, 994.500033578516], [0, 0, 1, 0], [0, 0, 0, 0], [9E9, 9E9, 9E9, 9E9, 9E9, 9E9]];
    CONST robtarget p4553:= [[1444.455182302372, 5.587550401036353, 994.500033578516], [0, 0, 1, 0], [0, 0, 0, 0], [9E9, 9E9, 9E9, 9E9, 9E9, 9E9]];
    CONST robtarget p4554:= [[1444.4897039717528, 5.9606160089632425, 994.500033578516], [0, 0, 1, 0], [0, 0, 0, 0], [9E9, 9E9, 9E9, 9E9, 9E9, 9E9]];
    CONST robtarget p4555:= [[1444.5709892191906, 6.6452162973559155, 994.500033578516], [0, 0, 1, 0], [0, 0, 0, 0], [9E9, 9E9, 9E9, 9E9, 9E9, 9E9]];
    CONST robtarget p4556:= [[1444.625081228523, 7.176420843300434, 994.500033578516], [0, 0, 1, 0], [0, 0, 0, 0], [9E9, 9E9, 9E9, 9E9, 9E9, 9E9]];
    CONST robtarget p4557:= [[1444.678954199502, 7.681099659551904, 994.500033578516], [0, 0, 1, 0], [0, 0, 0, 0], [9E9, 9E9, 9E9, 9E9, 9E9, 9E9]];
    CONST robtarget p4558:= [[1444.7250492582189, 8.027450103897337, 994.500033578516], [0, 0, 1, 0], [0, 0, 0, 0], [9E9, 9E9, 9E9, 9E9, 9E9, 9E9]];
    CONST robtarget p4559:= [[1444.7661030359684, 8.32719455435759, 994.500033578516], [0, 0, 1, 0], [0, 0, 0, 0], [9E9, 9E9, 9E9, 9E9, 9E9, 9E9]];
    CONST robtarget p4560:= [[1444.849709830874, 8.770763917857238, 994.500033578516], [0, 0, 1, 0], [0, 0, 0, 0], [9E9, 9E9, 9E9, 9E9, 9E9, 9E9]];
    CONST robtarget p4561:= [[1444.8955556767644, 9.024994806947731, 994.500033578516], [0, 0, 1, 0], [0, 0, 0, 0], [9E9, 9E9, 9E9, 9E9, 9E9, 9E9]];
    CONST robtarget p4562:= [[1444.9087428565897, 9.110494684914215, 994.500033578516], [0, 0, 1, 0], [0, 0, 0, 0], [9E9, 9E9, 9E9, 9E9, 9E9, 9E9]];
    CONST robtarget p4563:= [[1445.0081264117325, 9.648022136096259, 994.500033578516], [0, 0, 1, 0], [0, 0, 0, 0], [9E9, 9E9, 9E9, 9E9, 9E9, 9E9]];
    CONST robtarget p4564:= [[1445.0891864723746, 9.991241358546404, 994.500033578516], [0, 0, 1, 0], [0, 0, 0, 0], [9E9, 9E9, 9E9, 9E9, 9E9, 9E9]];
    CONST robtarget p4565:= [[1445.1608056532255, 10.455544457389209, 994.500033578516], [0, 0, 1, 0], [0, 0, 0, 0], [9E9, 9E9, 9E9, 9E9, 9E9, 9E9]];
    CONST robtarget p4566:= [[1445.2280483505403, 10.832812881088756, 994.500033578516], [0, 0, 1, 0], [0, 0, 0, 0], [9E9, 9E9, 9E9, 9E9, 9E9, 9E9]];
    CONST robtarget p4567:= [[1445.3273026202903, 11.334594288154292, 994.500033578516], [0, 0, 1, 0], [0, 0, 0, 0], [9E9, 9E9, 9E9, 9E9, 9E9, 9E9]];
    CONST robtarget p4568:= [[1445.3691119606065, 11.584701054371877, 994.500033578516], [0, 0, 1, 0], [0, 0, 0, 0], [9E9, 9E9, 9E9, 9E9, 9E9, 9E9]];
    CONST robtarget p4569:= [[1445.4051969002337, 11.750290374718716, 994.500033578516], [0, 0, 1, 0], [0, 0, 0, 0], [9E9, 9E9, 9E9, 9E9, 9E9, 9E9]];
    CONST robtarget p4570:= [[1445.4906176148809, 12.136469844422763, 994.500033578516], [0, 0, 1, 0], [0, 0, 0, 0], [9E9, 9E9, 9E9, 9E9, 9E9, 9E9]];
    CONST robtarget p4571:= [[1445.5624806736803, 12.4720839659865, 994.500033578516], [0, 0, 1, 0], [0, 0, 0, 0], [9E9, 9E9, 9E9, 9E9, 9E9, 9E9]];
    CONST robtarget p4572:= [[1445.5762265144053, 12.514151410589207, 994.500033578516], [0, 0, 1, 0], [0, 0, 0, 0], [9E9, 9E9, 9E9, 9E9, 9E9, 9E9]];
    CONST robtarget p4573:= [[1445.7413212505194, 13.153743720144234, 994.500033578516], [0, 0, 1, 0], [0, 0, 0, 0], [9E9, 9E9, 9E9, 9E9, 9E9, 9E9]];
    CONST robtarget p4574:= [[1445.7655227720718, 13.274309844829148, 994.500033578516], [0, 0, 1, 0], [0, 0, 0, 0], [9E9, 9E9, 9E9, 9E9, 9E9, 9E9]];
    CONST robtarget p4575:= [[1445.8211285690468, 13.475347406879749, 994.500033578516], [0, 0, 1, 0], [0, 0, 0, 0], [9E9, 9E9, 9E9, 9E9, 9E9, 9E9]];
    CONST robtarget p4576:= [[1445.9185459654461, 13.844176578579564, 994.500033578516], [0, 0, 1, 0], [0, 0, 0, 0], [9E9, 9E9, 9E9, 9E9, 9E9, 9E9]];
    CONST robtarget p4577:= [[1446.0525393785838, 14.34881838880753, 994.500033578516], [0, 0, 1, 0], [0, 0, 0, 0], [9E9, 9E9, 9E9, 9E9, 9E9, 9E9]];
    CONST robtarget p4578:= [[1446.0768973269985, 14.469847032011856, 994.500033578516], [0, 0, 1, 0], [0, 0, 0, 0], [9E9, 9E9, 9E9, 9E9, 9E9, 9E9]];
    CONST robtarget p4579:= [[1446.0787690422694, 14.477147669416553, 994.500033578516], [0, 0, 1, 0], [0, 0, 0, 0], [9E9, 9E9, 9E9, 9E9, 9E9, 9E9]];
    CONST robtarget p4580:= [[1446.1067905295135, 14.583932059985258, 994.500033578516], [0, 0, 1, 0], [0, 0, 0, 0], [9E9, 9E9, 9E9, 9E9, 9E9, 9E9]];
    CONST robtarget p4581:= [[1446.299700479995, 15.295300441874758, 994.500033578516], [0, 0, 1, 0], [0, 0, 0, 0], [9E9, 9E9, 9E9, 9E9, 9E9, 9E9]];
    CONST robtarget p4582:= [[1446.3602068791001, 15.513074305160913, 994.500033578516], [0, 0, 1, 0], [0, 0, 0, 0], [9E9, 9E9, 9E9, 9E9, 9E9, 9E9]];
    CONST robtarget p4583:= [[1446.4347206706684, 15.816277517954632, 994.500033578516], [0, 0, 1, 0], [0, 0, 0, 0], [9E9, 9E9, 9E9, 9E9, 9E9, 9E9]];
    CONST robtarget p4584:= [[1446.531686813625, 16.150514065965126, 994.500033578516], [0, 0, 1, 0], [0, 0, 0, 0], [9E9, 9E9, 9E9, 9E9, 9E9, 9E9]];
    CONST robtarget p4585:= [[1446.580819869369, 16.319014265025714, 994.500033578516], [0, 0, 1, 0], [0, 0, 0, 0], [9E9, 9E9, 9E9, 9E9, 9E9, 9E9]];
    CONST robtarget p4586:= [[1446.7943370339137, 16.883023358993043, 994.500033578516], [0, 0, 1, 0], [0, 0, 0, 0], [9E9, 9E9, 9E9, 9E9, 9E9, 9E9]];
    CONST robtarget p4587:= [[1446.8919010572313, 17.210122616875296, 994.500033578516], [0, 0, 1, 0], [0, 0, 0, 0], [9E9, 9E9, 9E9, 9E9, 9E9, 9E9]];
    CONST robtarget p4588:= [[1447.1089554992952, 17.866030268566348, 994.500033578516], [0, 0, 1, 0], [0, 0, 0, 0], [9E9, 9E9, 9E9, 9E9, 9E9, 9E9]];
    CONST robtarget p4589:= [[1447.322400080016, 18.491654992949805, 994.500033578516], [0, 0, 1, 0], [0, 0, 0, 0], [9E9, 9E9, 9E9, 9E9, 9E9, 9E9]];
    CONST robtarget p4590:= [[1447.4659540523473, 18.903860264407726, 994.500033578516], [0, 0, 1, 0], [0, 0, 0, 0], [9E9, 9E9, 9E9, 9E9, 9E9, 9E9]];
    CONST robtarget p4591:= [[1447.5447821413852, 19.115496570572105, 994.500033578516], [0, 0, 1, 0], [0, 0, 0, 0], [9E9, 9E9, 9E9, 9E9, 9E9, 9E9]];
    CONST robtarget p4592:= [[1447.6076232041391, 19.28292344683861, 994.500033578516], [0, 0, 1, 0], [0, 0, 0, 0], [9E9, 9E9, 9E9, 9E9, 9E9, 9E9]];
    CONST robtarget p4593:= [[1447.8049317873658, 19.903250404758978, 994.500033578516], [0, 0, 1, 0], [0, 0, 0, 0], [9E9, 9E9, 9E9, 9E9, 9E9, 9E9]];
    CONST robtarget p4594:= [[1447.8969791727604, 20.09699293191052, 994.500033578516], [0, 0, 1, 0], [0, 0, 0, 0], [9E9, 9E9, 9E9, 9E9, 9E9, 9E9]];
    CONST robtarget p4595:= [[1448.0609063464533, 20.500710034849902, 994.500033578516], [0, 0, 1, 0], [0, 0, 0, 0], [9E9, 9E9, 9E9, 9E9, 9E9, 9E9]];
    CONST robtarget p4596:= [[1448.2253810402433, 20.88937443912127, 994.500033578516], [0, 0, 1, 0], [0, 0, 0, 0], [9E9, 9E9, 9E9, 9E9, 9E9, 9E9]];
    CONST robtarget p4597:= [[1448.5048982169174, 21.534384219883492, 994.500033578516], [0, 0, 1, 0], [0, 0, 0, 0], [9E9, 9E9, 9E9, 9E9, 9E9, 9E9]];
    CONST robtarget p4598:= [[1448.5516458877348, 21.66400858080887, 994.500033578516], [0, 0, 1, 0], [0, 0, 0, 0], [9E9, 9E9, 9E9, 9E9, 9E9, 9E9]];
    CONST robtarget p4599:= [[1448.6286288891392, 21.839472791233305, 994.500033578516], [0, 0, 1, 0], [0, 0, 0, 0], [9E9, 9E9, 9E9, 9E9, 9E9, 9E9]];
    CONST robtarget p4600:= [[1448.761403422296, 22.1674068468122, 994.500033578516], [0, 0, 1, 0], [0, 0, 0, 0], [9E9, 9E9, 9E9, 9E9, 9E9, 9E9]];
    CONST robtarget p4601:= [[1449.0359672131594, 22.811136072658385, 994.500033578516], [0, 0, 1, 0], [0, 0, 0, 0], [9E9, 9E9, 9E9, 9E9, 9E9, 9E9]];
    CONST robtarget p4602:= [[1449.0999028437218, 22.969512727832196, 994.500033578516], [0, 0, 1, 0], [0, 0, 0, 0], [9E9, 9E9, 9E9, 9E9, 9E9, 9E9]];
    CONST robtarget p4603:= [[1449.1766993822173, 23.13856522266397, 994.500033578516], [0, 0, 1, 0], [0, 0, 0, 0], [9E9, 9E9, 9E9, 9E9, 9E9, 9E9]];
    CONST robtarget p4604:= [[1449.3018218305829, 23.419466140580184, 994.500033578516], [0, 0, 1, 0], [0, 0, 0, 0], [9E9, 9E9, 9E9, 9E9, 9E9, 9E9]];
    CONST robtarget p4605:= [[1449.40189348593, 23.668785356334098, 994.500033578516], [0, 0, 1, 0], [0, 0, 0, 0], [9E9, 9E9, 9E9, 9E9, 9E9, 9E9]];
    CONST robtarget p4606:= [[1449.5855518192725, 24.03655247762903, 994.500033578516], [0, 0, 1, 0], [0, 0, 0, 0], [9E9, 9E9, 9E9, 9E9, 9E9, 9E9]];
    CONST robtarget p4607:= [[1449.7735991453885, 24.40385430976599, 994.500033578516], [0, 0, 1, 0], [0, 0, 0, 0], [9E9, 9E9, 9E9, 9E9, 9E9, 9E9]];
    CONST robtarget p4608:= [[1449.797137028153, 24.445212726784206, 994.500033578516], [0, 0, 1, 0], [0, 0, 0, 0], [9E9, 9E9, 9E9, 9E9, 9E9, 9E9]];
    CONST robtarget p4609:= [[1450.0250733777186, 24.896247126409378, 994.500033578516], [0, 0, 1, 0], [0, 0, 0, 0], [9E9, 9E9, 9E9, 9E9, 9E9, 9E9]];
    CONST robtarget p4610:= [[1450.2497406622679, 25.333340627704032, 994.500033578516], [0, 0, 1, 0], [0, 0, 0, 0], [9E9, 9E9, 9E9, 9E9, 9E9, 9E9]];
    CONST robtarget p4611:= [[1450.2863397387532, 25.396437780867373, 994.500033578516], [0, 0, 1, 0], [0, 0, 0, 0], [9E9, 9E9, 9E9, 9E9, 9E9, 9E9]];
    CONST robtarget p4612:= [[1450.5700960861484, 25.932913360514036, 994.500033578516], [0, 0, 1, 0], [0, 0, 0, 0], [9E9, 9E9, 9E9, 9E9, 9E9, 9E9]];
    CONST robtarget p4613:= [[1450.6005634892856, 25.995152915707237, 994.500033578516], [0, 0, 1, 0], [0, 0, 0, 0], [9E9, 9E9, 9E9, 9E9, 9E9, 9E9]];
    CONST robtarget p4614:= [[1450.845114250685, 26.489512462606143, 994.500033578516], [0, 0, 1, 0], [0, 0, 0, 0], [9E9, 9E9, 9E9, 9E9, 9E9, 9E9]];
    CONST robtarget p4615:= [[1451.1983302391177, 27.168436467455763, 994.500033578516], [0, 0, 1, 0], [0, 0, 0, 0], [9E9, 9E9, 9E9, 9E9, 9E9, 9E9]];
    CONST robtarget p4616:= [[1451.532849394989, 27.74153615654734, 994.500033578516], [0, 0, 1, 0], [0, 0, 0, 0], [9E9, 9E9, 9E9, 9E9, 9E9, 9E9]];
    CONST robtarget p4617:= [[1451.7660220180062, 28.12609246522277, 994.500033578516], [0, 0, 1, 0], [0, 0, 0, 0], [9E9, 9E9, 9E9, 9E9, 9E9, 9E9]];
    CONST robtarget p4618:= [[1451.8297040291582, 28.23070226459687, 994.500033578516], [0, 0, 1, 0], [0, 0, 0, 0], [9E9, 9E9, 9E9, 9E9, 9E9, 9E9]];
    CONST robtarget p4619:= [[1451.980435252729, 28.47133240227477, 994.500033578516], [0, 0, 1, 0], [0, 0, 0, 0], [9E9, 9E9, 9E9, 9E9, 9E9, 9E9]];
    CONST robtarget p4620:= [[1452.1342159286198, 28.709965553042764, 994.500033578516], [0, 0, 1, 0], [0, 0, 0, 0], [9E9, 9E9, 9E9, 9E9, 9E9, 9E9]];
    CONST robtarget p4621:= [[1452.211684884929, 28.841325727736745, 994.500033578516], [0, 0, 1, 0], [0, 0, 0, 0], [9E9, 9E9, 9E9, 9E9, 9E9, 9E9]];
    CONST robtarget p4622:= [[1452.2789223386476, 28.954380522231403, 994.500033578516], [0, 0, 1, 0], [0, 0, 0, 0], [9E9, 9E9, 9E9, 9E9, 9E9, 9E9]];
    CONST robtarget p4623:= [[1452.3581223387177, 29.074390759419742, 994.500033578516], [0, 0, 1, 0], [0, 0, 0, 0], [9E9, 9E9, 9E9, 9E9, 9E9, 9E9]];
    CONST robtarget p4624:= [[1452.4836208100203, 29.281375282899702, 994.500033578516], [0, 0, 1, 0], [0, 0, 0, 0], [9E9, 9E9, 9E9, 9E9, 9E9, 9E9]];
    CONST robtarget p4625:= [[1452.5316159850395, 29.364989993557387, 994.500033578516], [0, 0, 1, 0], [0, 0, 0, 0], [9E9, 9E9, 9E9, 9E9, 9E9, 9E9]];
    CONST robtarget p4626:= [[1452.6789542284807, 29.622227471024047, 994.500033578516], [0, 0, 1, 0], [0, 0, 0, 0], [9E9, 9E9, 9E9, 9E9, 9E9, 9E9]];
    CONST robtarget p4627:= [[1452.736578404284, 29.72062287420134, 994.500033578516], [0, 0, 1, 0], [0, 0, 0, 0], [9E9, 9E9, 9E9, 9E9, 9E9, 9E9]];
    CONST robtarget p4628:= [[1452.7798822051486, 29.792437641699635, 994.500033578516], [0, 0, 1, 0], [0, 0, 0, 0], [9E9, 9E9, 9E9, 9E9, 9E9, 9E9]];
    CONST robtarget p4629:= [[1452.8140743440817, 29.8490437311045, 994.500033578516], [0, 0, 1, 0], [0, 0, 0, 0], [9E9, 9E9, 9E9, 9E9, 9E9, 9E9]];
    CONST robtarget p4630:= [[1453.1738126971559, 30.42476120294974, 994.500033578516], [0, 0, 1, 0], [0, 0, 0, 0], [9E9, 9E9, 9E9, 9E9, 9E9, 9E9]];
    CONST robtarget p4631:= [[1453.2998663907447, 30.641483779343915, 994.500033578516], [0, 0, 1, 0], [0, 0, 0, 0], [9E9, 9E9, 9E9, 9E9, 9E9, 9E9]];
    CONST robtarget p4632:= [[1453.6107235719344, 31.108226597382583, 994.500033578516], [0, 0, 1, 0], [0, 0, 0, 0], [9E9, 9E9, 9E9, 9E9, 9E9, 9E9]];
    CONST robtarget p4633:= [[1453.8584313610766, 31.447645790118315, 994.500033578516], [0, 0, 1, 0], [0, 0, 0, 0], [9E9, 9E9, 9E9, 9E9, 9E9, 9E9]];
    CONST robtarget p4634:= [[1453.9955737215032, 31.639361714682607, 994.500033578516], [0, 0, 1, 0], [0, 0, 0, 0], [9E9, 9E9, 9E9, 9E9, 9E9, 9E9]];
    CONST robtarget p4635:= [[1454.2490630306681, 31.994710634023903, 994.500033578516], [0, 0, 1, 0], [0, 0, 0, 0], [9E9, 9E9, 9E9, 9E9, 9E9, 9E9]];
    CONST robtarget p4636:= [[1454.5972480839532, 32.464287021853806, 994.500033578516], [0, 0, 1, 0], [0, 0, 0, 0], [9E9, 9E9, 9E9, 9E9, 9E9, 9E9]];
    CONST robtarget p4637:= [[1454.6410513735777, 32.52234140221371, 994.500033578516], [0, 0, 1, 0], [0, 0, 0, 0], [9E9, 9E9, 9E9, 9E9, 9E9, 9E9]];
    CONST robtarget p4638:= [[1454.9450251293972, 32.968547197336946, 994.500033578516], [0, 0, 1, 0], [0, 0, 0, 0], [9E9, 9E9, 9E9, 9E9, 9E9, 9E9]];
    CONST robtarget p4639:= [[1455.044555346359, 33.100775591106085, 994.500033578516], [0, 0, 1, 0], [0, 0, 0, 0], [9E9, 9E9, 9E9, 9E9, 9E9, 9E9]];
    CONST robtarget p4640:= [[1455.0956968928467, 33.164678580245905, 994.500033578516], [0, 0, 1, 0], [0, 0, 0, 0], [9E9, 9E9, 9E9, 9E9, 9E9, 9E9]];
    CONST robtarget p4641:= [[1455.3252649825138, 33.469513061241, 994.500033578516], [0, 0, 1, 0], [0, 0, 0, 0], [9E9, 9E9, 9E9, 9E9, 9E9, 9E9]];
    CONST robtarget p4642:= [[1455.6779575383143, 33.990628434736394, 994.500033578516], [0, 0, 1, 0], [0, 0, 0, 0], [9E9, 9E9, 9E9, 9E9, 9E9, 9E9]];
    CONST robtarget p4643:= [[1455.7427117386542, 34.0741015164577, 994.500033578516], [0, 0, 1, 0], [0, 0, 0, 0], [9E9, 9E9, 9E9, 9E9, 9E9, 9E9]];
    CONST robtarget p4644:= [[1456.002813878282, 34.40775737978112, 994.500033578516], [0, 0, 1, 0], [0, 0, 0, 0], [9E9, 9E9, 9E9, 9E9, 9E9, 9E9]];
    CONST robtarget p4645:= [[1456.0473616455365, 34.4618202050398, 994.500033578516], [0, 0, 1, 0], [0, 0, 0, 0], [9E9, 9E9, 9E9, 9E9, 9E9, 9E9]];
    CONST robtarget p4646:= [[1456.4684121899563, 34.95238369766078, 994.500033578516], [0, 0, 1, 0], [0, 0, 0, 0], [9E9, 9E9, 9E9, 9E9, 9E9, 9E9]];
    CONST robtarget p4647:= [[1456.563589290749, 35.06455908301977, 994.500033578516], [0, 0, 1, 0], [0, 0, 0, 0], [9E9, 9E9, 9E9, 9E9, 9E9, 9E9]];
    CONST robtarget p4648:= [[1456.6231206709988, 35.134540306802435, 994.500033578516], [0, 0, 1, 0], [0, 0, 0, 0], [9E9, 9E9, 9E9, 9E9, 9E9, 9E9]];
    CONST robtarget p4649:= [[1456.7700014899058, 35.31677548608185, 994.500033578516], [0, 0, 1, 0], [0, 0, 0, 0], [9E9, 9E9, 9E9, 9E9, 9E9, 9E9]];
    CONST robtarget p4650:= [[1457.0495309459768, 35.645030521683395, 994.500033578516], [0, 0, 1, 0], [0, 0, 0, 0], [9E9, 9E9, 9E9, 9E9, 9E9, 9E9]];
    CONST robtarget p4651:= [[1457.2661076605298, 35.92514365978023, 994.500033578516], [0, 0, 1, 0], [0, 0, 0, 0], [9E9, 9E9, 9E9, 9E9, 9E9, 9E9]];
    CONST robtarget p4652:= [[1457.2830556062768, 35.94454795718592, 994.500033578516], [0, 0, 1, 0], [0, 0, 0, 0], [9E9, 9E9, 9E9, 9E9, 9E9, 9E9]];
    CONST robtarget p4653:= [[1457.4228851314879, 36.112160470043506, 994.500033578516], [0, 0, 1, 0], [0, 0, 0, 0], [9E9, 9E9, 9E9, 9E9, 9E9, 9E9]];
    CONST robtarget p4654:= [[1457.511866427097, 36.218514801992555, 994.500033578516], [0, 0, 1, 0], [0, 0, 0, 0], [9E9, 9E9, 9E9, 9E9, 9E9, 9E9]];
    CONST robtarget p4655:= [[1457.7447786456453, 36.491851212374215, 994.500033578516], [0, 0, 1, 0], [0, 0, 0, 0], [9E9, 9E9, 9E9, 9E9, 9E9, 9E9]];
    CONST robtarget p4656:= [[1458.0435115676908, 36.860264177668654, 994.500033578516], [0, 0, 1, 0], [0, 0, 0, 0], [9E9, 9E9, 9E9, 9E9, 9E9, 9E9]];
    CONST robtarget p4657:= [[1458.573688416193, 37.463281098301664, 994.500033578516], [0, 0, 1, 0], [0, 0, 0, 0], [9E9, 9E9, 9E9, 9E9, 9E9, 9E9]];
    CONST robtarget p4658:= [[1458.7117828375044, 37.599402482521796, 994.500033578516], [0, 0, 1, 0], [0, 0, 0, 0], [9E9, 9E9, 9E9, 9E9, 9E9, 9E9]];
    CONST robtarget p4659:= [[1459.1354064166005, 38.045538494105415, 994.500033578516], [0, 0, 1, 0], [0, 0, 0, 0], [9E9, 9E9, 9E9, 9E9, 9E9, 9E9]];
    CONST robtarget p4660:= [[1459.2300569782901, 38.1456295436018, 994.500033578516], [0, 0, 1, 0], [0, 0, 0, 0], [9E9, 9E9, 9E9, 9E9, 9E9, 9E9]];
    CONST robtarget p4661:= [[1459.4505225409907, 38.374257948889564, 994.500033578516], [0, 0, 1, 0], [0, 0, 0, 0], [9E9, 9E9, 9E9, 9E9, 9E9, 9E9]];
    CONST robtarget p4662:= [[1459.5741103338335, 38.50374613226258, 994.500033578516], [0, 0, 1, 0], [0, 0, 0, 0], [9E9, 9E9, 9E9, 9E9, 9E9, 9E9]];
    CONST robtarget p4663:= [[1459.9445796052084, 38.88221115599012, 994.500033578516], [0, 0, 1, 0], [0, 0, 0, 0], [9E9, 9E9, 9E9, 9E9, 9E9, 9E9]];
    CONST robtarget p4664:= [[1460.121134895081, 39.06982162996431, 994.500033578516], [0, 0, 1, 0], [0, 0, 0, 0], [9E9, 9E9, 9E9, 9E9, 9E9, 9E9]];
    CONST robtarget p4665:= [[1460.5886630181378, 39.55729943489182, 994.500033578516], [0, 0, 1, 0], [0, 0, 0, 0], [9E9, 9E9, 9E9, 9E9, 9E9, 9E9]];
    CONST robtarget p4666:= [[1460.905445553548, 39.86850614091017, 994.500033578516], [0, 0, 1, 0], [0, 0, 0, 0], [9E9, 9E9, 9E9, 9E9, 9E9, 9E9]];
    CONST robtarget p4667:= [[1461.0483817779077, 40.00793701382119, 994.500033578516], [0, 0, 1, 0], [0, 0, 0, 0], [9E9, 9E9, 9E9, 9E9, 9E9, 9E9]];
    CONST robtarget p4668:= [[1461.347883697033, 40.30232480111883, 994.500033578516], [0, 0, 1, 0], [0, 0, 0, 0], [9E9, 9E9, 9E9, 9E9, 9E9, 9E9]];
    CONST robtarget p4669:= [[1461.721889044752, 40.65520999012476, 994.500033578516], [0, 0, 1, 0], [0, 0, 0, 0], [9E9, 9E9, 9E9, 9E9, 9E9, 9E9]];
    CONST robtarget p4670:= [[1461.974136980773, 40.873563807598586, 994.500033578516], [0, 0, 1, 0], [0, 0, 0, 0], [9E9, 9E9, 9E9, 9E9, 9E9, 9E9]];
    CONST robtarget p4671:= [[1462.1954729598551, 41.07416028457385, 994.500033578516], [0, 0, 1, 0], [0, 0, 0, 0], [9E9, 9E9, 9E9, 9E9, 9E9, 9E9]];
    CONST robtarget p4672:= [[1462.561366364617, 41.39160067345446, 994.500033578516], [0, 0, 1, 0], [0, 0, 0, 0], [9E9, 9E9, 9E9, 9E9, 9E9, 9E9]];
    CONST robtarget p4673:= [[1462.6461896734033, 41.47464154237568, 994.500033578516], [0, 0, 1, 0], [0, 0, 0, 0], [9E9, 9E9, 9E9, 9E9, 9E9, 9E9]];
    CONST robtarget p4674:= [[1462.8415331598735, 41.65022184133312, 994.500033578516], [0, 0, 1, 0], [0, 0, 0, 0], [9E9, 9E9, 9E9, 9E9, 9E9, 9E9]];
    CONST robtarget p4675:= [[1463.1824499321635, 41.96706751601543, 994.500033578516], [0, 0, 1, 0], [0, 0, 0, 0], [9E9, 9E9, 9E9, 9E9, 9E9, 9E9]];
    CONST robtarget p4676:= [[1463.385693985102, 42.14828817408775, 994.500033578516], [0, 0, 1, 0], [0, 0, 0, 0], [9E9, 9E9, 9E9, 9E9, 9E9, 9E9]];
    CONST robtarget p4677:= [[1463.520283380386, 42.264186844469634, 994.500033578516], [0, 0, 1, 0], [0, 0, 0, 0], [9E9, 9E9, 9E9, 9E9, 9E9, 9E9]];
    CONST robtarget p4678:= [[1463.6813645674101, 42.40575907673487, 994.500033578516], [0, 0, 1, 0], [0, 0, 0, 0], [9E9, 9E9, 9E9, 9E9, 9E9, 9E9]];
    CONST robtarget p4679:= [[1463.9917086838805, 42.67839602199261, 994.500033578516], [0, 0, 1, 0], [0, 0, 0, 0], [9E9, 9E9, 9E9, 9E9, 9E9, 9E9]];
    CONST robtarget p4680:= [[1464.1004424348578, 42.78364708516931, 994.500033578516], [0, 0, 1, 0], [0, 0, 0, 0], [9E9, 9E9, 9E9, 9E9, 9E9, 9E9]];
    CONST robtarget p4681:= [[1464.273959309511, 42.942444761300024, 994.500033578516], [0, 0, 1, 0], [0, 0, 0, 0], [9E9, 9E9, 9E9, 9E9, 9E9, 9E9]];
    CONST robtarget p4682:= [[1464.4234576613271, 43.05562125805321, 994.500033578516], [0, 0, 1, 0], [0, 0, 0, 0], [9E9, 9E9, 9E9, 9E9, 9E9, 9E9]];
